       // Shuttle 2
       "DB_OPC_Machine".Parameters.Presence.Shuttle2UndrilledPart := "DB_PartManagement".sPosition.sShuttle2.Undrilled.Presence.Part;
       "DB_OPC_Machine".Parameters.Presence.Shuttle2UndrilledBw := "DB_PartManagement".sPosition.sShuttle2.Undrilled.Presence.BW;
       "DB_OPC_Machine".Parameters.Presence.Shuttle2DrilledPart := "DB_PartManagement".sPosition.sShuttle2.Drilled.Presence.Part;
       "DB_OPC_Machine".Parameters.Presence.Shuttle2DrilledBw := "DB_PartManagement".sPosition.sShuttle2.Drilled.Presence.BW;

       // Gripper
       "DB_OPC_Machine".Parameters.Presence.GripperUndrilledPart := "DB_PartManagement".sPosition.sGripper.Undrilled.Presence.Part;
       "DB_OPC_Machine".Parameters.Presence.GripperUndrilledBw := "DB_PartManagement".sPosition.sGripper.Undrilled.Presence.BW;
       "DB_OPC_Machine".Parameters.Presence.GripperDrilledPart := "DB_PartManagement".sPosition.sGripper.Drilled.Presence.Part;
       "DB_OPC_Machine".Parameters.Presence.GripperDrilledBw := "DB_PartManagement".sPosition.sGripper.Drilled.Presence.BW;

       // Fixture
       "DB_OPC_Machine".Parameters.Presence.FixtureUndrilledPart := "DB_PartManagement".sPosition.sFixture.Undrilled.Presence.Part;
       "DB_OPC_Machine".Parameters.Presence.FixtureUndrilledBw := "DB_PartManagement".sPosition.sFixture.Undrilled.Presence.BW;
       "DB_OPC_Machine".Parameters.Presence.FixtureDrilledPart := "DB_PartManagement".sPosition.sFixture.Drilled.Presence.Part;
       "DB_OPC_Machine".Parameters.Presence.FixtureDrilledBw := "DB_PartManagement".sPosition.sFixture.Drilled.Presence.BW;
   END_REGION

   REGION Presence V2
       // // Shuttle 1
       // #sPresenceShuttle1UndrilledPart("HMI_Change Enable" := #sHmiChangeEnable,
       //                                 ioPLC_State := "DB_PartManagement".sPosition.sShuttle1.Undrilled.Presence.Part,
       //                                 ioHMI_State := "DB_OPC_Machine".Parameters.Presence.Shuttle1UndrilledPart);

       // #sPresenceShuttle1UndrilledBw("HMI_Change Enable" := #sHmiChangeEnable,
       //                               ioPLC_State := "DB_PartManagement".sPosition.sShuttle1.Undrilled.Presence.BW,
       //                               ioHMI_State := "DB_OPC_Machine".Parameters.Presence.Shuttle1UndrilledBw);

       // #sPresenceShuttle1DrilledPart("HMI_Change Enable" := #sHmiChangeEnable,
       //                                 ioPLC_State := "DB_PartManagement".sPosition.sShuttle1.Drilled.Presence.Part,
       //                                 ioHMI_State := "DB_OPC_Machine".Parameters.Presence.Shuttle1DrilledPart);

       // #sPresenceShuttle1DrilledBw("HMI_Change Enable" := #sHmiChangeEnable,
       //                               ioPLC_State := "DB_PartManagement".sPosition.sShuttle1.Drilled.Presence.BW,
       //                               ioHMI_State := "DB_OPC_Machine".Parameters.Presence.Shuttle1DrilledBw);

       //  // Shuttle 2
       //  #sPresenceShuttle2UndrilledPart("HMI_Change Enable" := #sHmiChangeEnable,
       //                                  ioPLC_State := "DB_PartManagement".sPosition.sShuttle2.Undrilled.Presence.Part,
       //                                  ioHMI_State := "DB_OPC_Machine".Parameters.Presence.Shuttle2UndrilledPart);

       //  #sPresenceShuttle2UndrilledBw("HMI_Change Enable" := #sHmiChangeEnable,
       //                                ioPLC_State := "DB_PartManagement".sPosition.sShuttle2.Undrilled.Presence.BW,
       //                                ioHMI_State := "DB_OPC_Machine".Parameters.Presence.Shuttle2UndrilledBw);

       //  #sPresenceShuttle2DrilledPart("HMI_Change Enable" := #sHmiChangeEnable,
       //                                ioPLC_State := "DB_PartManagement".sPosition.sShuttle2.Drilled.Presence.Part,
       //                                ioHMI_State := "DB_OPC_Machine".Parameters.Presence.Shuttle2DrilledPart);

       //  #sPresenceShuttle2DrilledBw("HMI_Change Enable" := #sHmiChangeEnable,
       //                              ioPLC_State := "DB_PartManagement".sPosition.sShuttle2.Drilled.Presence.BW,
       //                              ioHMI_State := "DB_OPC_Machine".Parameters.Presence.Shuttle2DrilledBw);

       //  // Gripper
       //  #sPresenceGripperUndrilledPart("HMI_Change Enable" := #sHmiChangeEnable,
       //                                 ioPLC_State := "DB_PartManagement".sPosition.sGripper.Undrilled.Presence.Part,
       //                                 ioHMI_State := "DB_OPC_Machine".Parameters.Presence.GripperUndrilledPart);

       //  #sPresenceGripperUndrilledBw("HMI_Change Enable" := #sHmiChangeEnable,
       //                               ioPLC_State := "DB_PartManagement".sPosition.sGripper.Undrilled.Presence.BW,
       //                               ioHMI_State := "DB_OPC_Machine".Parameters.Presence.GripperUndrilledBw);

       //  #sPresenceGripperDrilledPart("HMI_Change Enable" := #sHmiChangeEnable,
       //                               ioPLC_State := "DB_PartManagement".sPosition.sGripper.Drilled.Presence.Part,
       //                               ioHMI_State := "DB_OPC_Machine".Parameters.Presence.GripperDrilledPart);

       //  #sPresenceGripperDrilledBw("HMI_Change Enable" := #sHmiChangeEnable,
       //                             ioPLC_State := "DB_PartManagement".sPosition.sGripper.Drilled.Presence.BW,
       //                             ioHMI_State := "DB_OPC_Machine".Parameters.Presence.GripperDrilledBw);

       //  // Fixture
       //  #sPresenceFixtureUndrilledPart("HMI_Change Enable" := #sHmiChangeEnable,
       //                                 ioPLC_State := "DB_PartManagement".sPosition.sFixture.Undrilled.Presence.Part,
       //                                 ioHMI_State := "DB_OPC_Machine".Parameters.Presence.FixtureUndrilledPart);

       //  #sPresenceFixtureUndrilledBw("HMI_Change Enable" := #sHmiChangeEnable,
       //                               ioPLC_State := "DB_PartManagement".sPosition.sFixture.Undrilled.Presence.BW,
       //                               ioHMI_State := "DB_OPC_Machine".Parameters.Presence.FixtureUndrilledBw);

       //  #sPresenceFixtureDrilledPart("HMI_Change Enable" := #sHmiChangeEnable,
       //                               ioPLC_State := "DB_PartManagement".sPosition.sFixture.Drilled.Presence.Part,
       //                               ioHMI_State := "DB_OPC_Machine".Parameters.Presence.FixtureDrilledPart);

       //  #sPresenceFixtureDrilledBw("HMI_Change Enable" := #sHmiChangeEnable,
       //                             ioPLC_State := "DB_PartManagement".sPosition.sFixture.Drilled.Presence.BW,
       //                             ioHMI_State := "DB_OPC_Machine".Parameters.Presence.FixtureDrilledBw);
   END_REGION
END_FUNCTION_BLOCK

FUNCTION_BLOCK "FB_HMI_PLC_Pos"   // FB80, SCL
{ S7_Optimized_Access := 'TRUE' }
// stored: MemoryReserve 100, SetENOAutomatically false
   VAR_INPUT
      "HMI_Change Enable" : Bool;
   END_VAR
   VAR_IN_OUT
      ioPLC_State : Bool;
      ioHMI_State : Bool;
   END_VAR
   VAR
      PLC_StateMemo : Bool;
      HMI_StateMemo : Bool;
   END_VAR
BEGIN
   REGION Description header 
       //==================================================================================
       // POSALUX Swiss SA / (C) Copyright 2026
       //----------------------------------------------------------------------------------
       // Title: FB_HMI_PLC_Pos
       // Comment/Function: 
       // Author: Fabien WALDT
       // Engineering: TIA Portal v20
       //----------------------------------------------------------------------------------
       // Change log table:
       // Version  | Date     | Expert in charge | Changes applied
       // ---------|----------|------------------|-----------------------------------------
       // 00.00.01 | 20260521 | WFA              | First released version
       // =================================================================================
   END_REGION

   REGION Update Values
       IF #ioPLC_State <> #PLC_StateMemo OR NOT #"HMI_Change Enable" THEN
           #ioHMI_State := #ioPLC_State;
           #HMI_StateMemo := #ioPLC_State;
           #PLC_StateMemo := #ioPLC_State;
       ELSIF (#ioHMI_State <> #HMI_StateMemo) AND #"HMI_Change Enable" THEN
           #ioPLC_State := #ioHMI_State;
           #PLC_StateMemo := #ioHMI_State;
           #HMI_StateMemo := #ioHMI_State;
       END_IF;

   END_REGION
END_FUNCTION_BLOCK

FUNCTION_BLOCK "FB_OPC_AxisManagement"   // FB60, SCL
{ S7_Optimized_Access := 'TRUE' }
// stored: MemoryReserve 100, SetENOAutomatically false
   VAR
      sTeachButton : "FB_HmiKeysSignals";
      sAxisToTeachIndex { S7_SetPoint := 'True'} : DInt;
      sPositionToTeachIndex : DInt;
      sError { ExternalAccessible := 'False'; ExternalVisible := 'False'; ExternalWritable := 'False'} : Bool;
      sDone { ExternalAccessible := 'False'; ExternalVisible := 'False'; ExternalWritable := 'False'} : Bool;
      sState { ExternalAccessible := 'False'; ExternalVisible := 'False'; ExternalWritable := 'False'} : Word;
      sReadGUD_X_Load : "LBP_ReadGUD";
      sReadGUD_X_Unload { S7_SetPoint := 'True'} : "LBP_ReadGUD";
      sReadGUD_X_Blowing { S7_SetPoint := 'True'} : "LBP_ReadGUD";
      sReadGUD_Y_Load : "LBP_ReadGUD";
      sReadGUD_Y_Unload { S7_SetPoint := 'True'} : "LBP_ReadGUD";
      sReadGUD_Y_Blowing { S7_SetPoint := 'True'} : "LBP_ReadGUD";
      sReadGUD_B_Load : "LBP_ReadGUD";
      sReadGUD_B_Unload { S7_SetPoint := 'True'} : "LBP_ReadGUD";
      sReadGUD_B_Blowing { S7_SetPoint := 'True'} : "LBP_ReadGUD";
      sReadGUD_ZM_Safe { S7_SetPoint := 'True'} : "LBP_ReadGUD";
      sReadGUD_ZL_Safe { S7_SetPoint := 'True'} : "LBP_ReadGUD";
      sVarName { S7_SetPoint := 'True'} : String;
      sTON_On : TON_TIME;
      sTON_OFF { S7_SetPoint := 'True'} : TON_TIME;
      sPulseReadGUD { S7_SetPoint := 'True'} : Bool;
      sID : Int;
   END_VAR
   VAR_TEMP
      tIndex : Int;
   END_VAR
   VAR CONSTANT
      U1_AXIS_ID : DInt := 111;
      U2_AXIS_ID : DInt := 112;
      V_AXIS_ID : DInt := 120;
      W_AXIS_ID : DInt := 130;
      X_AXIS_ID : DInt := 210;
      Y_AXIS_ID : DInt := 220;
      ZL_AXIS_ID : DInt := 230;
      ZM_AXIS_ID : DInt := 240;
      B_AXIS_ID : DInt := 320;
      EXTERNAL_LOADER_ID : DInt := 211;
      SEMI_AUTO_ID : DInt := 212;
      EXT_OF_SAFETY_GATE_EXT_ID : DInt := 221;
      INT_OF_SAFETY_GATE_EXT_ID : DInt := 222;
      INSIDE_SAFETY_GATE_ID : DInt := 223;
      EXT_OF_SAFETY_GATE_INT_ID : DInt := 224;
      INT_OF_SAFETY_GATE_INT_ID : DInt := 225;
      PART_DETECTOR_ID : DInt := 230;
      BACKWALL_LOAD_ID : DInt := 241;
      BACKWALL_UNLOAD_ID : DInt := 242;
      BACKWALL_DETECTOR_ID : DInt := 250;
      LOADER_BLOW_TO_SHUTTLE_ID : DInt := 260;
      LOADER_BLOW_TO_SHUTTLE_1_ID : DInt := 261;
      LOADER_BLOW_TO_SHUTTLE_2_ID : DInt := 262;
      FROM_SHUTTLE_TO_LOADER_ID : DInt := 310;
      FROM_SHUTTLE_1_TO_LOADER : DInt := 311;
      FROM_SHUTTLE_2_TO_LOADER : DInt := 312;
      SAFE : DInt := 400;
      APPROACH_SHUTTLE_1 : DInt := 421;
      APPROACH_SHUTTLE_2 : DInt := 422;
      APPROACH_WORK_CLAMP : DInt := 430;
      FROM_LOADER_TO_WORK : DInt := 610;
      FROM_WORK_TO_LOADER : DInt := 620;
      LOADER_BLOW_TO_WORK : DInt := 730;
      STATION1 : Byte := 1;
   END_VAR
BEGIN
   REGION Description header 
       //==================================================================================
       // POSALUX Swiss SA / (C) Copyright 2025
       //----------------------------------------------------------------------------------
       // Title: FB_OPC_AxisManagement
       // Comment/Function: 
       // Author: Fabien WALDT
       // Engineering: TIA Portal v20
       //----------------------------------------------------------------------------------
       // Change log table:
       // Version  | Date     | Expert in charge | Changes applied
       // ---------|----------|------------------|-----------------------------------------
       // 00.00.01 | 20260109 | WFA              | First released version
       // =================================================================================
   END_REGION
   REGION Axis - Actual Values
       // Number of axis
       "DB_OPC_Axis".ActualValues.NumberOfAxes := 9;

       // Axis01_X
       #sID := 1;
       "DB_OPC_Axis".ActualValues.Axes[#sID].ActualPosition := "DB_AxisPosition".sAxis01_X."$AA_IM";
       "DB_OPC_Axis".ActualValues.Axes[#sID].AxisId := #X_AXIS_ID;
       "DB_OPC_Axis".ActualValues.Axes[#sID].StationNumber := #STATION1;
       // Axis02_Y
       #sID := #sID + 1;
       "DB_OPC_Axis".ActualValues.Axes[#sID].ActualPosition := "DB_AxisPosition".sAxis02_Y."$AA_IM";
       "DB_OPC_Axis".ActualValues.Axes[#sID].AxisId := #Y_AXIS_ID;
       "DB_OPC_Axis".ActualValues.Axes[#sID].StationNumber := #STATION1;
       // Axis03_ZM
       #sID := #sID + 1;
       "DB_OPC_Axis".ActualValues.Axes[#sID].ActualPosition := "DB_AxisPosition".sAxis03_ZM."$AA_IM";
       "DB_OPC_Axis".ActualValues.Axes[#sID].AxisId := #ZM_AXIS_ID;
       "DB_OPC_Axis".ActualValues.Axes[#sID].StationNumber := #STATION1;
       // Axis04_B
       #sID := #sID + 1;
       "DB_OPC_Axis".ActualValues.Axes[#sID].ActualPosition := "DB_AxisPosition".sAxis04_B."$AA_IM";
       "DB_OPC_Axis".ActualValues.Axes[#sID].AxisId := #B_AXIS_ID;
       "DB_OPC_Axis".ActualValues.Axes[#sID].StationNumber := #STATION1;
       // Axis05_U1
       #sID := #sID + 1;
       "DB_OPC_Axis".ActualValues.Axes[#sID].ActualPosition := "DB_AxisPosition".sAxis05_U1."$AA_IM";
       "DB_OPC_Axis".ActualValues.Axes[#sID].AxisId := #U1_AXIS_ID;
       "DB_OPC_Axis".ActualValues.Axes[#sID].StationNumber := #STATION1;
       // Axis06_U2
       #sID := #sID + 1;
       "DB_OPC_Axis".ActualValues.Axes[#sID].ActualPosition := "DB_AxisPosition".sAxis06_U2."$AA_IM";
       "DB_OPC_Axis".ActualValues.Axes[#sID].AxisId := #U2_AXIS_ID;
       "DB_OPC_Axis".ActualValues.Axes[#sID].StationNumber := #STATION1;
       // Axis07_V
       #sID := #sID + 1;
       "DB_OPC_Axis".ActualValues.Axes[#sID].ActualPosition := "DB_AxisPosition".sAxis07_V."$AA_IM";
       "DB_OPC_Axis".ActualValues.Axes[#sID].AxisId := #V_AXIS_ID;
       "DB_OPC_Axis".ActualValues.Axes[#sID].StationNumber := #STATION1;
       // Axis08_W
       #sID := #sID + 1;
       "DB_OPC_Axis".ActualValues.Axes[#sID].ActualPosition := "DB_AxisPosition".sAxis08_W."$AA_IM";
       "DB_OPC_Axis".ActualValues.Axes[#sID].AxisId := #W_AXIS_ID;
       "DB_OPC_Axis".ActualValues.Axes[#sID].StationNumber := #STATION1;
       // Axis09_ZL
       #sID := #sID + 1;
       "DB_OPC_Axis".ActualValues.Axes[#sID].ActualPosition := "DB_AxisPosition".sAxis09_ZL."$AA_IM";
       "DB_OPC_Axis".ActualValues.Axes[#sID].AxisId := #ZL_AXIS_ID;
       "DB_OPC_Axis".ActualValues.Axes[#sID].StationNumber := #STATION1;
   END_REGION

   REGION Taught Position PLC
       // Number of items
       "DB_OPC_Axis".TaughtPositions.NumberOfItems := 48;

       REGION Axis05_U1
           // External loader
           #sID := 1;
           "DB_OPC_Axis".TaughtPositions.Items[#sID].AxisId := #U1_AXIS_ID;
           "DB_OPC_Axis".TaughtPositions.Items[#sID].PositionId := #EXTERNAL_LOADER_ID;
           "DB_OPC_Axis".TaughtPositions.Items[#sID].StationNumber := #STATION1;
           "DB_OPC_Axis".TaughtPositions.Items[#sID].Value := "DB_AxisPosMachinePLC".Axis_U1.ExtLoadUnloadAuto;
           // Semi-auto
           #sID := #sID + 1;
           "DB_OPC_Axis".TaughtPositions.Items[#sID].AxisId := #U1_AXIS_ID;
           "DB_OPC_Axis".TaughtPositions.Items[#sID].PositionId := #SEMI_AUTO_ID;
           "DB_OPC_Axis".TaughtPositions.Items[#sID].StationNumber := #STATION1;
           "DB_OPC_Axis".TaughtPositions.Items[#sID].Value := "DB_AxisPosMachinePLC".Axis_U1.ExtLoadUnloadManu;
           // Ext of safety gate ext
           #sID := #sID + 1;
           "DB_OPC_Axis".TaughtPositions.Items[#sID].AxisId := #U1_AXIS_ID;
           "DB_OPC_Axis".TaughtPositions.Items[#sID].PositionId := #EXT_OF_SAFETY_GATE_EXT_ID;
           "DB_OPC_Axis".TaughtPositions.Items[#sID].StationNumber := #STATION1;
           "DB_OPC_Axis".TaughtPositions.Items[#sID].Value := "DB_AxisPosMachinePLC".Axis_U1.ExtGateExt;
           // Int of safety gate ext
           #sID := #sID + 1;
           "DB_OPC_Axis".TaughtPositions.Items[#sID].AxisId := #U1_AXIS_ID;
           "DB_OPC_Axis".TaughtPositions.Items[#sID].PositionId := #INT_OF_SAFETY_GATE_EXT_ID;
           "DB_OPC_Axis".TaughtPositions.Items[#sID].StationNumber := #STATION1;
           "DB_OPC_Axis".TaughtPositions.Items[#sID].Value := "DB_AxisPosMachinePLC".Axis_U1.IntGateExt;
           // Inside safety gate
           #sID := #sID + 1;
           "DB_OPC_Axis".TaughtPositions.Items[#sID].AxisId := #U1_AXIS_ID;
           "DB_OPC_Axis".TaughtPositions.Items[#sID].PositionId := #INSIDE_SAFETY_GATE_ID;
           "DB_OPC_Axis".TaughtPositions.Items[#sID].StationNumber := #STATION1;
           "DB_OPC_Axis".TaughtPositions.Items[#sID].Value := "DB_AxisPosMachinePLC".Axis_U1.Sas;
           // Ext of safety gate Int
           #sID := #sID + 1;
           "DB_OPC_Axis".TaughtPositions.Items[#sID].AxisId := #U1_AXIS_ID;
           "DB_OPC_Axis".TaughtPositions.Items[#sID].PositionId := #EXT_OF_SAFETY_GATE_INT_ID;
           "DB_OPC_Axis".TaughtPositions.Items[#sID].StationNumber := #STATION1;
           "DB_OPC_Axis".TaughtPositions.Items[#sID].Value := "DB_AxisPosMachinePLC".Axis_U1.ExtGateInt;
           // Int of safety gate Int
           #sID := #sID + 1;
           "DB_OPC_Axis".TaughtPositions.Items[#sID].AxisId := #U1_AXIS_ID;
           "DB_OPC_Axis".TaughtPositions.Items[#sID].PositionId := #INT_OF_SAFETY_GATE_INT_ID;
           "DB_OPC_Axis".TaughtPositions.Items[#sID].StationNumber := #STATION1;
           "DB_OPC_Axis".TaughtPositions.Items[#sID].Value := "DB_AxisPosMachinePLC".Axis_U1.IntGateInt;
           // Part detector
           #sID := #sID + 1;
           "DB_OPC_Axis".TaughtPositions.Items[#sID].AxisId := #U1_AXIS_ID;
           "DB_OPC_Axis".TaughtPositions.Items[#sID].PositionId := #PART_DETECTOR_ID;
           "DB_OPC_Axis".TaughtPositions.Items[#sID].StationNumber := #STATION1;
           "DB_OPC_Axis".TaughtPositions.Items[#sID].Value := "DB_AxisPosMachinePLC".Axis_U1.PartControl;
           // Backwall load
           #sID := #sID + 1;
           "DB_OPC_Axis".TaughtPositions.Items[#sID].AxisId := #U1_AXIS_ID;
           "DB_OPC_Axis".TaughtPositions.Items[#sID].PositionId := #BACKWALL_LOAD_ID;
           "DB_OPC_Axis".TaughtPositions.Items[#sID].StationNumber := #STATION1;
           "DB_OPC_Axis".TaughtPositions.Items[#sID].Value := "DB_AxisPosMachinePLC".Axis_U1.BwLoad;
           // Backwall unload
           #sID := #sID + 1;
           "DB_OPC_Axis".TaughtPositions.Items[#sID].AxisId := #U1_AXIS_ID;
           "DB_OPC_Axis".TaughtPositions.Items[#sID].PositionId := #BACKWALL_UNLOAD_ID;
           "DB_OPC_Axis".TaughtPositions.Items[#sID].StationNumber := #STATION1;
           "DB_OPC_Axis".TaughtPositions.Items[#sID].Value := "DB_AxisPosMachinePLC".Axis_U1.BwUnLoad;
           // Backwall detector
           #sID := #sID + 1;
           "DB_OPC_Axis".TaughtPositions.Items[#sID].AxisId := #U1_AXIS_ID;
           "DB_OPC_Axis".TaughtPositions.Items[#sID].PositionId := #BACKWALL_DETECTOR_ID;
           "DB_OPC_Axis".TaughtPositions.Items[#sID].StationNumber := #STATION1;
           "DB_OPC_Axis".TaughtPositions.Items[#sID].Value := "DB_AxisPosMachinePLC".Axis_U1.BwControl;
           // Loader blow to shuttle
           #sID := #sID + 1;
           "DB_OPC_Axis".TaughtPositions.Items[#sID].AxisId := #U1_AXIS_ID;
           "DB_OPC_Axis".TaughtPositions.Items[#sID].PositionId := #LOADER_BLOW_TO_SHUTTLE_ID;
           "DB_OPC_Axis".TaughtPositions.Items[#sID].StationNumber := #STATION1;
           "DB_OPC_Axis".TaughtPositions.Items[#sID].Value := "DB_AxisPosMachinePLC".Axis_U1.Blowing;
           // From shuttle to Loader
           #sID := #sID + 1;
           "DB_OPC_Axis".TaughtPositions.Items[#sID].AxisId := #U1_AXIS_ID;
           "DB_OPC_Axis".TaughtPositions.Items[#sID].PositionId := #FROM_SHUTTLE_TO_LOADER_ID;
           "DB_OPC_Axis".TaughtPositions.Items[#sID].StationNumber := #STATION1;
           "DB_OPC_Axis".TaughtPositions.Items[#sID].Value := "DB_AxisPosMachinePLC".Axis_U1.IntLoadUnload;
       END_REGION

       REGION Axis06_U2
           // External loader
           #sID := #sID + 1;
           "DB_OPC_Axis".TaughtPositions.Items[#sID].AxisId := #U2_AXIS_ID;
           "DB_OPC_Axis".TaughtPositions.Items[#sID].PositionId := #EXTERNAL_LOADER_ID;
           "DB_OPC_Axis".TaughtPositions.Items[#sID].StationNumber := #STATION1;
           "DB_OPC_Axis".TaughtPositions.Items[#sID].Value := "DB_AxisPosMachinePLC".Axis_U2.ExtLoadUnloadAuto;
           // Semi-auto
           #sID := #sID + 1;
           "DB_OPC_Axis".TaughtPositions.Items[#sID].AxisId := #U2_AXIS_ID;
           "DB_OPC_Axis".TaughtPositions.Items[#sID].PositionId := #SEMI_AUTO_ID;
           "DB_OPC_Axis".TaughtPositions.Items[#sID].StationNumber := #STATION1;
           "DB_OPC_Axis".TaughtPositions.Items[#sID].Value := "DB_AxisPosMachinePLC".Axis_U2.ExtLoadUnloadManu;
           // Ext of safety gate ext
           #sID := #sID + 1;
           "DB_OPC_Axis".TaughtPositions.Items[#sID].AxisId := #U2_AXIS_ID;
           "DB_OPC_Axis".TaughtPositions.Items[#sID].PositionId := #EXT_OF_SAFETY_GATE_EXT_ID;
           "DB_OPC_Axis".TaughtPositions.Items[#sID].StationNumber := #STATION1;
           "DB_OPC_Axis".TaughtPositions.Items[#sID].Value := "DB_AxisPosMachinePLC".Axis_U2.ExtGateExt;
           // Int of safety gate ext
           #sID := #sID + 1;
           "DB_OPC_Axis".TaughtPositions.Items[#sID].AxisId := #U2_AXIS_ID;
           "DB_OPC_Axis".TaughtPositions.Items[#sID].PositionId := #INT_OF_SAFETY_GATE_EXT_ID;
           "DB_OPC_Axis".TaughtPositions.Items[#sID].StationNumber := #STATION1;
           "DB_OPC_Axis".TaughtPositions.Items[#sID].Value := "DB_AxisPosMachinePLC".Axis_U2.IntGateExt;
           // Inside safety gate
           #sID := #sID + 1;
           "DB_OPC_Axis".TaughtPositions.Items[#sID].AxisId := #U2_AXIS_ID;
           "DB_OPC_Axis".TaughtPositions.Items[#sID].PositionId := #INSIDE_SAFETY_GATE_ID;
           "DB_OPC_Axis".TaughtPositions.Items[#sID].StationNumber := #STATION1;
           "DB_OPC_Axis".TaughtPositions.Items[#sID].Value := "DB_AxisPosMachinePLC".Axis_U2.Sas;
           // Ext of safety gate Int
           #sID := #sID + 1;
           "DB_OPC_Axis".TaughtPositions.Items[#sID].AxisId := #U2_AXIS_ID;
           "DB_OPC_Axis".TaughtPositions.Items[#sID].PositionId := #EXT_OF_SAFETY_GATE_INT_ID;
           "DB_OPC_Axis".TaughtPositions.Items[#sID].StationNumber := #STATION1;
           "DB_OPC_Axis".TaughtPositions.Items[#sID].Value := "DB_AxisPosMachinePLC".Axis_U2.ExtGateInt;
           // Int of safety gate Int
           #sID := #sID + 1;
           "DB_OPC_Axis".TaughtPositions.Items[#sID].AxisId := #U2_AXIS_ID;
           "DB_OPC_Axis".TaughtPositions.Items[#sID].PositionId := #INT_OF_SAFETY_GATE_INT_ID;
           "DB_OPC_Axis".TaughtPositions.Items[#sID].StationNumber := #STATION1;
           "DB_OPC_Axis".TaughtPositions.Items[#sID].Value := "DB_AxisPosMachinePLC".Axis_U2.IntGateInt;
           // Part detector
           #sID := #sID + 1;
           "DB_OPC_Axis".TaughtPositions.Items[#sID].AxisId := #U2_AXIS_ID;
           "DB_OPC_Axis".TaughtPositions.Items[#sID].PositionId := #PART_DETECTOR_ID;
           "DB_OPC_Axis".TaughtPositions.Items[#sID].StationNumber := #STATION1;
           "DB_OPC_Axis".TaughtPositions.Items[#sID].Value := "DB_AxisPosMachinePLC".Axis_U2.PartControl;
           // Backwall load
           #sID := #sID + 1;
           "DB_OPC_Axis".TaughtPositions.Items[#sID].AxisId := #U2_AXIS_ID;
           "DB_OPC_Axis".TaughtPositions.Items[#sID].PositionId := #BACKWALL_LOAD_ID;
           "DB_OPC_Axis".TaughtPositions.Items[#sID].StationNumber := #STATION1;
           "DB_OPC_Axis".TaughtPositions.Items[#sID].Value := "DB_AxisPosMachinePLC".Axis_U2.BwLoad;
           // Backwall unload
           #sID := #sID + 1;
           "DB_OPC_Axis".TaughtPositions.Items[#sID].AxisId := #U2_AXIS_ID;
           "DB_OPC_Axis".TaughtPositions.Items[#sID].PositionId := #BACKWALL_UNLOAD_ID;
           "DB_OPC_Axis".TaughtPositions.Items[#sID].StationNumber := #STATION1;
           "DB_OPC_Axis".TaughtPositions.Items[#sID].Value := "DB_AxisPosMachinePLC".Axis_U2.BwUnLoad;
           // Backwall detector
           #sID := #sID + 1;
           "DB_OPC_Axis".TaughtPositions.Items[#sID].AxisId := #U2_AXIS_ID;
           "DB_OPC_Axis".TaughtPositions.Items[#sID].PositionId := #BACKWALL_DETECTOR_ID;
           "DB_OPC_Axis".TaughtPositions.Items[#sID].StationNumber := #STATION1;
           "DB_OPC_Axis".TaughtPositions.Items[#sID].Value := "DB_AxisPosMachinePLC".Axis_U2.BwControl;
           // Loader blow to shuttle
           #sID := #sID + 1;
           "DB_OPC_Axis".TaughtPositions.Items[#sID].AxisId := #U2_AXIS_ID;
           "DB_OPC_Axis".TaughtPositions.Items[#sID].PositionId := #LOADER_BLOW_TO_SHUTTLE_ID;
           "DB_OPC_Axis".TaughtPositions.Items[#sID].StationNumber := #STATION1;
           "DB_OPC_Axis".TaughtPositions.Items[#sID].Value := "DB_AxisPosMachinePLC".Axis_U2.Blowing;
           // From shuttle to Loader
           #sID := #sID + 1;
           "DB_OPC_Axis".TaughtPositions.Items[#sID].AxisId := #U2_AXIS_ID;
           "DB_OPC_Axis".TaughtPositions.Items[#sID].PositionId := #FROM_SHUTTLE_TO_LOADER_ID;
           "DB_OPC_Axis".TaughtPositions.Items[#sID].StationNumber := #STATION1;
           "DB_OPC_Axis".TaughtPositions.Items[#sID].Value := "DB_AxisPosMachinePLC".Axis_U2.IntLoadUnload;
       END_REGION

       REGION Axis07_V
           // Loader blow to shuttle 1
           #sID := #sID + 1;
           "DB_OPC_Axis".TaughtPositions.Items[#sID].AxisId := #V_AXIS_ID;
           "DB_OPC_Axis".TaughtPositions.Items[#sID].PositionId := #LOADER_BLOW_TO_SHUTTLE_1_ID;
           "DB_OPC_Axis".TaughtPositions.Items[#sID].StationNumber := #STATION1;
           "DB_OPC_Axis".TaughtPositions.Items[#sID].Value := "DB_AxisPosMachinePLC".Axis_V.Shuttle_1.Blowing;
           // Loader blow to shuttle 2
           #sID := #sID + 1;
           "DB_OPC_Axis".TaughtPositions.Items[#sID].AxisId := #V_AXIS_ID;
           "DB_OPC_Axis".TaughtPositions.Items[#sID].PositionId := #LOADER_BLOW_TO_SHUTTLE_2_ID;
           "DB_OPC_Axis".TaughtPositions.Items[#sID].StationNumber := #STATION1;
           "DB_OPC_Axis".TaughtPositions.Items[#sID].Value := "DB_AxisPosMachinePLC".Axis_V.Shuttle_2.Blowing;
           // From shuttle 1 to loader
           #sID := #sID + 1;
           "DB_OPC_Axis".TaughtPositions.Items[#sID].AxisId := #V_AXIS_ID;
           "DB_OPC_Axis".TaughtPositions.Items[#sID].PositionId := #FROM_SHUTTLE_1_TO_LOADER;
           "DB_OPC_Axis".TaughtPositions.Items[#sID].StationNumber := #STATION1;
           "DB_OPC_Axis".TaughtPositions.Items[#sID].Value := "DB_AxisPosMachinePLC".Axis_V.Shuttle_1.LoadUnload;
           // From shuttle 2 to loader
           #sID := #sID + 1;
           "DB_OPC_Axis".TaughtPositions.Items[#sID].AxisId := #V_AXIS_ID;
           "DB_OPC_Axis".TaughtPositions.Items[#sID].PositionId := #FROM_SHUTTLE_2_TO_LOADER;
           "DB_OPC_Axis".TaughtPositions.Items[#sID].StationNumber := #STATION1;
           "DB_OPC_Axis".TaughtPositions.Items[#sID].Value := "DB_AxisPosMachinePLC".Axis_V.Shuttle_2.LoadUnload;
           // Safe
           #sID := #sID + 1;
           "DB_OPC_Axis".TaughtPositions.Items[#sID].AxisId := #V_AXIS_ID;
           "DB_OPC_Axis".TaughtPositions.Items[#sID].PositionId := #SAFE;
           "DB_OPC_Axis".TaughtPositions.Items[#sID].StationNumber := #STATION1;
           "DB_OPC_Axis".TaughtPositions.Items[#sID].Value := "DB_AxisPosMachinePLC".Axis_V.Safe;
       END_REGION

       REGION Axis08_W
           // Loader blow to shuttle 1
           #sID := #sID + 1;
           "DB_OPC_Axis".TaughtPositions.Items[#sID].AxisId := #W_AXIS_ID;
           "DB_OPC_Axis".TaughtPositions.Items[#sID].PositionId := #LOADER_BLOW_TO_SHUTTLE_1_ID;
           "DB_OPC_Axis".TaughtPositions.Items[#sID].StationNumber := #STATION1;
           "DB_OPC_Axis".TaughtPositions.Items[#sID].Value := "DB_AxisPosMachinePLC".Axis_W.Shuttle_1.Blowing;
           // Loader blow to shuttle 2
           #sID := #sID + 1;
           "DB_OPC_Axis".TaughtPositions.Items[#sID].AxisId := #W_AXIS_ID;
           "DB_OPC_Axis".TaughtPositions.Items[#sID].PositionId := #LOADER_BLOW_TO_SHUTTLE_2_ID;
           "DB_OPC_Axis".TaughtPositions.Items[#sID].StationNumber := #STATION1;
           "DB_OPC_Axis".TaughtPositions.Items[#sID].Value := "DB_AxisPosMachinePLC".Axis_W.Shuttle_2.Blowing;
           // From shuttle 1 to loader
           #sID := #sID + 1;
           "DB_OPC_Axis".TaughtPositions.Items[#sID].AxisId := #W_AXIS_ID;
           "DB_OPC_Axis".TaughtPositions.Items[#sID].PositionId := #FROM_SHUTTLE_1_TO_LOADER;
           "DB_OPC_Axis".TaughtPositions.Items[#sID].StationNumber := #STATION1;
           "DB_OPC_Axis".TaughtPositions.Items[#sID].Value := "DB_AxisPosMachinePLC".Axis_W.Shuttle_1.LoadUnload;
           // From shuttle 2 to loader
           #sID := #sID + 1;
           "DB_OPC_Axis".TaughtPositions.Items[#sID].AxisId := #W_AXIS_ID;
           "DB_OPC_Axis".TaughtPositions.Items[#sID].PositionId := #FROM_SHUTTLE_2_TO_LOADER;
           "DB_OPC_Axis".TaughtPositions.Items[#sID].StationNumber := #STATION1;
           "DB_OPC_Axis".TaughtPositions.Items[#sID].Value := "DB_AxisPosMachinePLC".Axis_W.Shuttle_2.LoadUnload;
           // Safe
           #sID := #sID + 1;
           "DB_OPC_Axis".TaughtPositions.Items[#sID].AxisId := #W_AXIS_ID;
           "DB_OPC_Axis".TaughtPositions.Items[#sID].PositionId := #SAFE;
           "DB_OPC_Axis".TaughtPositions.Items[#sID].StationNumber := #STATION1;
           "DB_OPC_Axis".TaughtPositions.Items[#sID].Value := "DB_AxisPosMachinePLC".Axis_W.Safe;
       END_REGION

       REGION Axis07_V (Fixture)
           // From loader to work
           #sID := #sID + 1;
           "DB_OPC_Axis".TaughtPositions.Items[#sID].AxisId := #V_AXIS_ID;
           "DB_OPC_Axis".TaughtPositions.Items[#sID].PositionId := #FROM_LOADER_TO_WORK;
           "DB_OPC_Axis".TaughtPositions.Items[#sID].StationNumber := #STATION1;
           "DB_OPC_Axis".TaughtPositions.Items[#sID].Value := "DB_AxisPosMachinePLC".Axis_V.Fixture.Load;
           // From work to loader
           #sID := #sID + 1;
           "DB_OPC_Axis".TaughtPositions.Items[#sID].AxisId := #V_AXIS_ID;
           "DB_OPC_Axis".TaughtPositions.Items[#sID].PositionId := #FROM_WORK_TO_LOADER;
           "DB_OPC_Axis".TaughtPositions.Items[#sID].StationNumber := #STATION1;
           "DB_OPC_Axis".TaughtPositions.Items[#sID].Value := "DB_AxisPosMachinePLC".Axis_V.Fixture.Unload;
           // Loader blow to work
           #sID := #sID + 1;
           "DB_OPC_Axis".TaughtPositions.Items[#sID].AxisId := #V_AXIS_ID;
           "DB_OPC_Axis".TaughtPositions.Items[#sID].PositionId := #LOADER_BLOW_TO_WORK;
           "DB_OPC_Axis".TaughtPositions.Items[#sID].StationNumber := #STATION1;
           "DB_OPC_Axis".TaughtPositions.Items[#sID].Value := "DB_AxisPosMachinePLC".Axis_V.Fixture.Blowing;
       END_REGION

       REGION Axis08_W (Fixture)
           // Approach work clamp NOT USED
           // #sID := #sID + 1;
           // "DB_OPC_Axis".TaughtPositions.Items[#sID].AxisId := #W_AXIS_ID;
           // "DB_OPC_Axis".TaughtPositions.Items[#sID].PositionId := #APPROACH_WORK_CLAMP;
           // "DB_OPC_Axis".TaughtPositions.Items[#sID].StationNumber := #STATION1;
           // "DB_OPC_Axis".TaughtPositions.Items[#sID].Value := "DB_AxisPosMachineNC".Axis_W.Approach;
           // From loader to work
           #sID := #sID + 1;
           "DB_OPC_Axis".TaughtPositions.Items[#sID].AxisId := #W_AXIS_ID;
           "DB_OPC_Axis".TaughtPositions.Items[#sID].PositionId := #FROM_LOADER_TO_WORK;
           "DB_OPC_Axis".TaughtPositions.Items[#sID].StationNumber := #STATION1;
           "DB_OPC_Axis".TaughtPositions.Items[#sID].Value := "DB_AxisPosMachinePLC".Axis_W.Fixture.Load;
           // From work to loader
           #sID := #sID + 1;
           "DB_OPC_Axis".TaughtPositions.Items[#sID].AxisId := #W_AXIS_ID;
           "DB_OPC_Axis".TaughtPositions.Items[#sID].PositionId := #FROM_WORK_TO_LOADER;
           "DB_OPC_Axis".TaughtPositions.Items[#sID].StationNumber := #STATION1;
           "DB_OPC_Axis".TaughtPositions.Items[#sID].Value := "DB_AxisPosMachinePLC".Axis_W.Fixture.Unload;
           // Loader blow to work
           #sID := #sID + 1;
           "DB_OPC_Axis".TaughtPositions.Items[#sID].AxisId := #W_AXIS_ID;
           "DB_OPC_Axis".TaughtPositions.Items[#sID].PositionId := #LOADER_BLOW_TO_WORK;
           "DB_OPC_Axis".TaughtPositions.Items[#sID].StationNumber := #STATION1;
           "DB_OPC_Axis".TaughtPositions.Items[#sID].Value := "DB_AxisPosMachinePLC".Axis_W.Fixture.Blowing;
       END_REGION
   END_REGION

   REGION Taught Position NC
       REGION Axis01_X
           // From loader to work
           #sID := #sID + 1;
           "DB_OPC_Axis".TaughtPositions.Items[#sID].AxisId := #X_AXIS_ID;
           "DB_OPC_Axis".TaughtPositions.Items[#sID].PositionId := #FROM_LOADER_TO_WORK;
           "DB_OPC_Axis".TaughtPositions.Items[#sID].StationNumber := #STATION1;
           "DB_OPC_Axis".TaughtPositions.Items[#sID].Value := "DB_AxisPosMachineNC".Axis_X.Load;
           // From work to loader
           #sID := #sID + 1;
           "DB_OPC_Axis".TaughtPositions.Items[#sID].AxisId := #X_AXIS_ID;
           "DB_OPC_Axis".TaughtPositions.Items[#sID].PositionId := #FROM_WORK_TO_LOADER;
           "DB_OPC_Axis".TaughtPositions.Items[#sID].StationNumber := #STATION1;
           "DB_OPC_Axis".TaughtPositions.Items[#sID].Value := "DB_AxisPosMachineNC".Axis_X.Unload;
           // Loader blow to work
           #sID := #sID + 1;
           "DB_OPC_Axis".TaughtPositions.Items[#sID].AxisId := #X_AXIS_ID;
           "DB_OPC_Axis".TaughtPositions.Items[#sID].PositionId := #LOADER_BLOW_TO_WORK;
           "DB_OPC_Axis".TaughtPositions.Items[#sID].StationNumber := #STATION1;
           "DB_OPC_Axis".TaughtPositions.Items[#sID].Value := "DB_AxisPosMachineNC".Axis_X.Blowing;
       END_REGION

       REGION Axis02_Y
           // From loader to work
           #sID := #sID + 1;
           "DB_OPC_Axis".TaughtPositions.Items[#sID].AxisId := #Y_AXIS_ID;
           "DB_OPC_Axis".TaughtPositions.Items[#sID].PositionId := #FROM_LOADER_TO_WORK;
           "DB_OPC_Axis".TaughtPositions.Items[#sID].StationNumber := #STATION1;
           "DB_OPC_Axis".TaughtPositions.Items[#sID].Value := "DB_AxisPosMachineNC".Axis_Y.Load;
           // From work to loader
           #sID := #sID + 1;
           "DB_OPC_Axis".TaughtPositions.Items[#sID].AxisId := #Y_AXIS_ID;
           "DB_OPC_Axis".TaughtPositions.Items[#sID].PositionId := #FROM_WORK_TO_LOADER;
           "DB_OPC_Axis".TaughtPositions.Items[#sID].StationNumber := #STATION1;
           "DB_OPC_Axis".TaughtPositions.Items[#sID].Value := "DB_AxisPosMachineNC".Axis_Y.Unload;
           // Loader blow to work
           #sID := #sID + 1;
           "DB_OPC_Axis".TaughtPositions.Items[#sID].AxisId := #Y_AXIS_ID;
           "DB_OPC_Axis".TaughtPositions.Items[#sID].PositionId := #LOADER_BLOW_TO_WORK;
           "DB_OPC_Axis".TaughtPositions.Items[#sID].StationNumber := #STATION1;
           "DB_OPC_Axis".TaughtPositions.Items[#sID].Value := "DB_AxisPosMachineNC".Axis_Y.Blowing;
       END_REGION

       // REGION Axis04_B Not Used
       //     // From loader to work
       //     #sID := #sID + 1;
       //     "DB_OPC_Axis".TaughtPositions.Items[#sID].AxisId := #B_AXIS_ID;
       //     "DB_OPC_Axis".TaughtPositions.Items[#sID].PositionId := #FROM_LOADER_TO_WORK;
       //     "DB_OPC_Axis".TaughtPositions.Items[#sID].StationNumber := #STATION1;
       //     "DB_OPC_Axis".TaughtPositions.Items[#sID].Value := "DB_AxisPosMachineNC".Axis_B.Load;
       //     // From work to loader
       //     #sID := #sID + 1;
       //     "DB_OPC_Axis".TaughtPositions.Items[#sID].AxisId := #B_AXIS_ID;
       //     "DB_OPC_Axis".TaughtPositions.Items[#sID].PositionId := #FROM_WORK_TO_LOADER;
       //     "DB_OPC_Axis".TaughtPositions.Items[#sID].StationNumber := #STATION1;
       //     "DB_OPC_Axis".TaughtPositions.Items[#sID].Value := "DB_AxisPosMachineNC".Axis_B.Unload;
       //     // Loader blow to work
       //     #sID := #sID + 1;
       //     "DB_OPC_Axis".TaughtPositions.Items[#sID].AxisId := #B_AXIS_ID;
       //     "DB_OPC_Axis".TaughtPositions.Items[#sID].PositionId := #LOADER_BLOW_TO_WORK;
       //     "DB_OPC_Axis".TaughtPositions.Items[#sID].StationNumber := #STATION1;
       //     "DB_OPC_Axis".TaughtPositions.Items[#sID].Value := "DB_AxisPosMachineNC".Axis_B.Blowing;
       // END_REGION


   END_REGION

   REGION Teach
       // Call button
       #sTeachButton(ioOPC := "DB_OPC_Axis".Teach.Buttons.Teach);
       #sTeachButton.sKeyDisable := "LBP_ModeGroup".E_JOG;
       #sTeachButton.sLedSWStatus := #sTeachButton.sKeySWToggleStatus;

       // Search axis index
       #sAxisToTeachIndex := 0;
       "DB_OPC_Axis".Teach.Current.ActualPosition := 0.0;
       FOR #tIndex := 1 TO "DB_OPC_Axis".ActualValues.NumberOfAxes DO
           IF "DB_OPC_Axis".ActualValues.Axes[#tIndex].AxisId = "DB_OPC_Axis".Teach.Parameters.AxisId THEN
               #sAxisToTeachIndex := #tIndex;
               "DB_OPC_Axis".Teach.Current.ActualPosition := "DB_OPC_Axis".ActualValues.Axes[#sAxisToTeachIndex].ActualPosition;
           END_IF;
       END_FOR;
       // Search position index
       #sPositionToTeachIndex := 0;
       "DB_OPC_Axis".Teach.Current.TaughtPosition := 0.0;
       FOR #tIndex := 1 TO "DB_OPC_Axis".TaughtPositions.NumberOfItems DO
           IF "DB_OPC_Axis".TaughtPositions.Items[#tIndex].AxisId = "DB_OPC_Axis".Teach.Parameters.AxisId
               AND "DB_OPC_Axis".TaughtPositions.Items[#tIndex].PositionId = "DB_OPC_Axis".Teach.Parameters.PositionId THEN
               #sPositionToTeachIndex := #tIndex;
               "DB_OPC_Axis".Teach.Current.TaughtPosition := "DB_OPC_Axis".TaughtPositions.Items[#sPositionToTeachIndex].Value;
           END_IF;
       END_FOR;

       // // If Teach Button, Copy Axis ActualPosition to TaughtPosition 
       // IF #TeachButton.KeySWToggleStatus THEN
       //     "DB_OPC_Axis".TaughtPositions.Items[#PositionToTeachIndex].Value := "DB_OPC_Axis".ActualValues.Axes[#AxisToTeachIndex].ActualPosition;
       //     #TeachButton.KeySWToggleStatus := FALSE;
       // END_IF;
   END_REGION

   REGION Copy Current values to Taught Values
       IF #sTeachButton.sKeySWToggleStatus THEN
           CASE "DB_OPC_Axis".Teach.Parameters.AxisId OF
           #U1_AXIS_ID:
               CASE "DB_OPC_Axis".Teach.Parameters.PositionId OF
                   #EXTERNAL_LOADER_ID:
                       "DB_AxisPosMachinePLC".Axis_U1.ExtLoadUnloadAuto := "DB_AxisPosition".sAxis05_U1."$AA_IM";
                   #SEMI_AUTO_ID:
                       "DB_AxisPosMachinePLC".Axis_U1.ExtLoadUnloadManu := "DB_AxisPosition".sAxis05_U1."$AA_IM";
                   #EXT_OF_SAFETY_GATE_EXT_ID:
                       "DB_AxisPosMachinePLC".Axis_U1.ExtGateExt := "DB_AxisPosition".sAxis05_U1."$AA_IM";
                   #INT_OF_SAFETY_GATE_EXT_ID:
                       "DB_AxisPosMachinePLC".Axis_U1.IntGateExt := "DB_AxisPosition".sAxis05_U1."$AA_IM";
                   #INSIDE_SAFETY_GATE_ID:
                       "DB_AxisPosMachinePLC".Axis_U1.Sas := "DB_AxisPosition".sAxis05_U1."$AA_IM";
                   #EXT_OF_SAFETY_GATE_INT_ID:
                       "DB_AxisPosMachinePLC".Axis_U1.ExtGateInt := "DB_AxisPosition".sAxis05_U1."$AA_IM";
                   #INT_OF_SAFETY_GATE_INT_ID:
                       "DB_AxisPosMachinePLC".Axis_U1.IntGateInt := "DB_AxisPosition".sAxis05_U1."$AA_IM";
                   #PART_DETECTOR_ID:
                       "DB_AxisPosMachinePLC".Axis_U1.PartControl := "DB_AxisPosition".sAxis05_U1."$AA_IM";
                   #BACKWALL_LOAD_ID:
                       "DB_AxisPosMachinePLC".Axis_U1.BwLoad := "DB_AxisPosition".sAxis05_U1."$AA_IM";
                   #BACKWALL_UNLOAD_ID:
                       "DB_AxisPosMachinePLC".Axis_U1.BwUnLoad := "DB_AxisPosition".sAxis05_U1."$AA_IM";
                   #BACKWALL_DETECTOR_ID:
                       "DB_AxisPosMachinePLC".Axis_U1.BwControl := "DB_AxisPosition".sAxis05_U1."$AA_IM";
                   #LOADER_BLOW_TO_SHUTTLE_ID:
                       "DB_AxisPosMachinePLC".Axis_U1.Blowing := "DB_AxisPosition".sAxis05_U1."$AA_IM";
                   #FROM_SHUTTLE_TO_LOADER_ID:
                       "DB_AxisPosMachinePLC".Axis_U1.IntLoadUnload := "DB_AxisPosition".sAxis05_U1."$AA_IM";
               END_CASE;
           #U2_AXIS_ID:
               CASE "DB_OPC_Axis".Teach.Parameters.PositionId OF
                   #EXTERNAL_LOADER_ID:
                       "DB_AxisPosMachinePLC".Axis_U1.ExtLoadUnloadAuto := "DB_AxisPosition".sAxis06_U2."$AA_IM";
                   #SEMI_AUTO_ID:
                       "DB_AxisPosMachinePLC".Axis_U1.ExtLoadUnloadManu := "DB_AxisPosition".sAxis06_U2."$AA_IM";
                   #EXT_OF_SAFETY_GATE_EXT_ID:
                       "DB_AxisPosMachinePLC".Axis_U1.ExtGateExt := "DB_AxisPosition".sAxis06_U2."$AA_IM";
                   #INT_OF_SAFETY_GATE_EXT_ID:
                       "DB_AxisPosMachinePLC".Axis_U1.IntGateExt := "DB_AxisPosition".sAxis06_U2."$AA_IM";
                   #INSIDE_SAFETY_GATE_ID:
                       "DB_AxisPosMachinePLC".Axis_U1.Sas := "DB_AxisPosition".sAxis06_U2."$AA_IM";
                   #EXT_OF_SAFETY_GATE_INT_ID:
                       "DB_AxisPosMachinePLC".Axis_U1.ExtGateInt := "DB_AxisPosition".sAxis06_U2."$AA_IM";
                   #INT_OF_SAFETY_GATE_INT_ID:
                       "DB_AxisPosMachinePLC".Axis_U1.IntGateInt := "DB_AxisPosition".sAxis06_U2."$AA_IM";
                   #PART_DETECTOR_ID:
                       "DB_AxisPosMachinePLC".Axis_U1.PartControl := "DB_AxisPosition".sAxis06_U2."$AA_IM";
                   #BACKWALL_LOAD_ID:
                       "DB_AxisPosMachinePLC".Axis_U1.BwLoad := "DB_AxisPosition".sAxis06_U2."$AA_IM";
                   #BACKWALL_UNLOAD_ID:
                       "DB_AxisPosMachinePLC".Axis_U1.BwUnLoad := "DB_AxisPosition".sAxis06_U2."$AA_IM";
                   #BACKWALL_DETECTOR_ID:
                       "DB_AxisPosMachinePLC".Axis_U1.BwControl := "DB_AxisPosition".sAxis06_U2."$AA_IM";
                   #LOADER_BLOW_TO_SHUTTLE_ID:
                       "DB_AxisPosMachinePLC".Axis_U1.Blowing := "DB_AxisPosition".sAxis06_U2."$AA_IM";
                   #FROM_SHUTTLE_TO_LOADER_ID:
                       "DB_AxisPosMachinePLC".Axis_U1.IntLoadUnload := "DB_AxisPosition".sAxis06_U2."$AA_IM";
               END_CASE;
           #V_AXIS_ID:
               CASE "DB_OPC_Axis".Teach.Parameters.PositionId OF
                   #LOADER_BLOW_TO_SHUTTLE_1_ID:
                       "DB_AxisPosMachinePLC".Axis_V.Shuttle_1.Blowing := "DB_AxisPosition".sAxis07_V."$AA_IM";
                   #LOADER_BLOW_TO_SHUTTLE_2_ID:
                       "DB_AxisPosMachinePLC".Axis_V.Shuttle_2.Blowing := "DB_AxisPosition".sAxis07_V."$AA_IM";
                   #FROM_SHUTTLE_1_TO_LOADER:
                       "DB_AxisPosMachinePLC".Axis_V.Shuttle_1.LoadUnload := "DB_AxisPosition".sAxis07_V."$AA_IM";
                   #FROM_SHUTTLE_2_TO_LOADER:
                       "DB_AxisPosMachinePLC".Axis_V.Shuttle_2.LoadUnload := "DB_AxisPosition".sAxis07_V."$AA_IM";
                   #SAFE:
                       "DB_AxisPosMachinePLC".Axis_V.Safe := "DB_AxisPosition".sAxis07_V."$AA_IM";

                   #FROM_LOADER_TO_WORK:
                       "DB_AxisPosMachinePLC".Axis_V.Fixture.Load := "DB_AxisPosition".sAxis07_V."$AA_IM";
                   #FROM_WORK_TO_LOADER:
                       "DB_AxisPosMachinePLC".Axis_V.Fixture.Unload := "DB_AxisPosition".sAxis07_V."$AA_IM";
                   #LOADER_BLOW_TO_WORK:
                       "DB_AxisPosMachinePLC".Axis_V.Fixture.Blowing := "DB_AxisPosition".sAxis07_V."$AA_IM";
               END_CASE;
           #W_AXIS_ID:
               CASE "DB_OPC_Axis".Teach.Parameters.PositionId OF
                   #LOADER_BLOW_TO_SHUTTLE_1_ID:
                       "DB_AxisPosMachinePLC".Axis_W.Shuttle_1.Blowing := "DB_AxisPosition".sAxis08_W."$AA_IM";
                   #LOADER_BLOW_TO_SHUTTLE_2_ID:
                       "DB_AxisPosMachinePLC".Axis_W.Shuttle_2.Blowing := "DB_AxisPosition".sAxis08_W."$AA_IM";
                   #FROM_SHUTTLE_1_TO_LOADER:
                       "DB_AxisPosMachinePLC".Axis_W.Shuttle_1.LoadUnload := "DB_AxisPosition".sAxis08_W."$AA_IM";
                   #FROM_SHUTTLE_2_TO_LOADER:
                       "DB_AxisPosMachinePLC".Axis_W.Shuttle_2.LoadUnload := "DB_AxisPosition".sAxis08_W."$AA_IM";
                   #SAFE:
                       "DB_AxisPosMachinePLC".Axis_W.Safe := "DB_AxisPosition".sAxis08_W."$AA_IM";

                   #FROM_LOADER_TO_WORK:
                       "DB_AxisPosMachinePLC".Axis_V.Fixture.Load := "DB_AxisPosition".sAxis08_W."$AA_IM";
                   #FROM_WORK_TO_LOADER:
                       "DB_AxisPosMachinePLC".Axis_V.Fixture.Unload := "DB_AxisPosition".sAxis08_W."$AA_IM";
                   #LOADER_BLOW_TO_WORK:
                       "DB_AxisPosMachinePLC".Axis_V.Fixture.Blowing := "DB_AxisPosition".sAxis08_W."$AA_IM";
               END_CASE;
           #X_AXIS_ID:
               CASE "DB_OPC_Axis".Teach.Parameters.PositionId OF
                   #FROM_LOADER_TO_WORK:
                       "DB_AxisPosMachineNC".Axis_X.Load := "DB_AxisPosition".sAxis01_X."$AA_IM";
                   #FROM_WORK_TO_LOADER:
                       "DB_AxisPosMachineNC".Axis_X.Unload := "DB_AxisPosition".sAxis01_X."$AA_IM";
                   #LOADER_BLOW_TO_WORK:
                       "DB_AxisPosMachineNC".Axis_X.Blowing := "DB_AxisPosition".sAxis01_X."$AA_IM";
               END_CASE;
           #Y_AXIS_ID:
               CASE "DB_OPC_Axis".Teach.Parameters.PositionId OF
                   #FROM_LOADER_TO_WORK:
                       "DB_AxisPosMachineNC".Axis_X.Load := "DB_AxisPosition".sAxis02_Y."$AA_IM";
                   #FROM_WORK_TO_LOADER:
                       "DB_AxisPosMachineNC".Axis_X.Unload := "DB_AxisPosition".sAxis02_Y."$AA_IM";
                   #LOADER_BLOW_TO_WORK:
                       "DB_AxisPosMachineNC".Axis_X.Blowing := "DB_AxisPosition".sAxis02_Y."$AA_IM";
               END_CASE;
           #B_AXIS_ID:
               CASE "DB_OPC_Axis".Teach.Parameters.PositionId OF
                   #FROM_LOADER_TO_WORK:
                       "DB_AxisPosMachineNC".Axis_X.Load := "DB_AxisPosition".sAxis04_B."$AA_IM";
                   #FROM_WORK_TO_LOADER:
                       "DB_AxisPosMachineNC".Axis_X.Unload := "DB_AxisPosition".sAxis04_B."$AA_IM";
                   #LOADER_BLOW_TO_WORK:
                       "DB_AxisPosMachineNC".Axis_X.Blowing := "DB_AxisPosition".sAxis04_B."$AA_IM";
               END_CASE;
       END_CASE;
       #sTeachButton.sKeySWToggleStatus := FALSE;
     END_IF;
   END_REGION

   REGION Read NC Position

       // TON phase ON (5 secondes)
       #sTON_On(
              IN := #sPulseReadGUD,
              PT := T#5s);

       // TON phase OFF (5 secondes)
       #sTON_OFF(
               IN := NOT #sPulseReadGUD,
               PT := T#5s);

      IF #sTON_On.Q THEN
           #sPulseReadGUD := FALSE;
       END_IF;

       IF #sTON_OFF.Q THEN
           #sPulseReadGUD := TRUE;
       END_IF;


       REGION X Axis
           #sVarName := 'CH_X_LOAD';

           #sReadGUD_X_Load(Req := #sPulseReadGUD,
                           Addr := #sVarName,
                           Area := 2,
                           Unit := 1,
                           Index1 := 0,
                           Index2 := 0,
                           CnvtToken := FALSE,
                           VarToken := NULL,
                           Error => #sReadGUD_X_Load.Error,
                           Done => #sReadGUD_X_Load.Done,
                           State => #sReadGUD_X_Load.State,
                           RD := "DB_AxisPosMachineNC".Axis_X.Load);

           #sVarName := 'CH_X_UNLOAD';

           #sReadGUD_X_Unload(Req := #sPulseReadGUD,
                           Addr := #sVarName,
                           Area := 2,
                           Unit := 1,
                           Index1 := 0,
                           Index2 := 0,
                           CnvtToken := FALSE,
                           VarToken := NULL,
                           Error => #sReadGUD_X_Unload.Error,
                           Done => #sReadGUD_X_Unload.Done,
                           State => #sReadGUD_X_Unload.State,
                           RD := "DB_AxisPosMachineNC".Axis_X.Unload);

           #sVarName := 'CH_X_BLOW';

           #sReadGUD_X_Blowing(Req := #sPulseReadGUD,
                                  Addr := #sVarName,
                                  Area := 2,
                                  Unit := 1,
                                  Index1 := 0,
                                  Index2 := 0,
                                  CnvtToken := FALSE,
                                  VarToken := NULL,
                                  Error => #sReadGUD_X_Blowing.Error,
                                  Done => #sReadGUD_X_Blowing.Done,
                                  State => #sReadGUD_X_Blowing.State,
                                  RD := "DB_AxisPosMachineNC".Axis_X.Blowing);
       END_REGION
       REGION Y Axis
           #sVarName := 'CH_Y_LOAD';

           #sReadGUD_Y_Load(Req := NOT #sPulseReadGUD,
                           Addr := #sVarName,
                           Area := 2,
                           Unit := 1,
                           Index1 := 0,
                           Index2 := 0,
                           CnvtToken := FALSE,
                           VarToken := NULL,
                           Error => #sReadGUD_Y_Load.Error,
                           Done => #sReadGUD_Y_Load.Done,
                           State => #sReadGUD_Y_Load.State,
                           RD := "DB_AxisPosMachineNC".Axis_Y.Load);

           #sVarName := 'CH_Y_UNLOAD';

           #sReadGUD_Y_Unload(Req := NOT #sPulseReadGUD,
                             Addr := #sVarName,
                             Area := 2,
                             Unit := 1,
                             Index1 := 0,
                             Index2 := 0,
                             CnvtToken := FALSE,
                             VarToken := NULL,
                             Error => #sReadGUD_Y_Unload.Error,
                             Done => #sReadGUD_Y_Unload.Done,
                             State => #sReadGUD_Y_Unload.State,
                             RD := "DB_AxisPosMachineNC".Axis_Y.Unload);

           #sVarName := 'CH_Y_BLOW';

           #sReadGUD_Y_Blowing(Req := NOT #sPulseReadGUD,
                              Addr := #sVarName,
                              Area := 2,
                              Unit := 1,
                              Index1 := 0,
                              Index2 := 0,
                              CnvtToken := FALSE,
                              VarToken := NULL,
                              Error => #sReadGUD_Y_Blowing.Error,
                              Done => #sReadGUD_Y_Blowing.Done,
                              State => #sReadGUD_Y_Blowing.State,
                              RD := "DB_AxisPosMachineNC".Axis_Y.Blowing);
       END_REGION
       REGION B Axis
           #sVarName := 'CH_B_LOAD';

           #sReadGUD_B_Load(Req := #sPulseReadGUD,
                           Addr := #sVarName,
                           Area := 2,
                           Unit := 1,
                           Index1 := 0,
                           Index2 := 0,
                           CnvtToken := FALSE,
                           VarToken := NULL,
                           Error => #sReadGUD_B_Load.Error,
                           Done => #sReadGUD_B_Load.Done,
                           State => #sReadGUD_B_Load.State,
                           RD := "DB_AxisPosMachineNC".Axis_B.Load);

           #sVarName := 'CH_B_UNLOAD';

           #sReadGUD_B_Unload(Req := #sPulseReadGUD,
                             Addr := #sVarName,
                             Area := 2,
                             Unit := 1,
                             Index1 := 0,
                             Index2 := 0,
                             CnvtToken := FALSE,
                             VarToken := NULL,
                             Error => #sReadGUD_B_Unload.Error,
                             Done => #sReadGUD_B_Unload.Done,
                             State => #sReadGUD_B_Unload.State,
                             RD := "DB_AxisPosMachineNC".Axis_B.Unload);

           #sVarName := 'CH_B_BLOW';

           #sReadGUD_B_Blowing(Req := #sPulseReadGUD,
                              Addr := #sVarName,
                              Area := 2,
                              Unit := 1,
                              Index1 := 0,
                              Index2 := 0,
                              CnvtToken := FALSE,
                              VarToken := NULL,
                              Error => #sReadGUD_B_Blowing.Error,
                              Done => #sReadGUD_B_Blowing.Done,
                              State => #sReadGUD_B_Blowing.State,
                              RD := "DB_AxisPosMachineNC".Axis_B.Blowing);
       END_REGION
       REGION ZM Axis
           #sVarName := 'CH_ZM_SAFE';

           #sReadGUD_ZM_Safe(Req := #sPulseReadGUD,
                              Addr := #sVarName,
                              Area := 2,
                              Unit := 1,
                              Index1 := 0,
                              Index2 := 0,
                              CnvtToken := FALSE,
                              VarToken := NULL,
                              Error => #sReadGUD_ZM_Safe.Error,
                              Done => #sReadGUD_ZM_Safe.Done,
                              State => #sReadGUD_ZM_Safe.State,
                              RD := "DB_AxisPosMachineNC".Axis_ZM.Safe);
         END_REGION

         REGION ZL Axis
             #sVarName := 'CH_ZL_SAFE';

             #sReadGUD_ZL_Safe(Req := NOT #sPulseReadGUD,
                              Addr := #sVarName,
                              Area := 2,
                              Unit := 1,
                              Index1 := 0,
                              Index2 := 0,
                              CnvtToken := FALSE,
                              VarToken := NULL,
                              Error => #sReadGUD_ZL_Safe.Error,
                              Done => #sReadGUD_ZL_Safe.Done,
                              State => #sReadGUD_ZL_Safe.State,
                              RD := "DB_AxisPosMachineNC".Axis_ZL.Safe);
         END_REGION
   END_REGION
END_FUNCTION_BLOCK

FUNCTION_BLOCK "FB_HmiKeysSignals"   // FB812, SCL
{ S7_Optimized_Access := 'TRUE' }
// stored: AutoNumber false, MemoryReserve 100, SetENOAutomatically false
   VAR_IN_OUT
      ioOPC : "UDT_OPC_Button";
   END_VAR
   VAR
      sKeySWStatus : Bool;
      sKeySWToggleStatus : Bool;
      sKeyDisable : Bool;
      sKeySWPositiveFront : Bool;
      sKeySWNegativeFront : Bool;
      sKeySWTogglePositiveFront : Bool;
      sKeySWToggleNegativeFront : Bool;
      sLedSWStatus : Bool;
      sLedSWStatusBlink : Bool;
      sRT_KeySWPositiveFront { S7_SetPoint := 'True'} : R_TRIG;
      sFT_KeySWNegativeFront { S7_SetPoint := 'True'} : F_TRIG;
      sRT_KeySWTogglePositiveFront { S7_SetPoint := 'True'} : R_TRIG;
      sFT_KeySWToggleNegativeFront { S7_SetPoint := 'True'} : F_TRIG;
   END_VAR
BEGIN
   REGION Description header 
       //==================================================================================
       // POSALUX Swiss SA / (C) Copyright 2025
       //----------------------------------------------------------------------------------
       // Title: FB_HmiKeysSignals 
       // Comment/Function: 
       //
       // Author: Fabien Waldt
       // Engineering: TIA Portal v19
       //----------------------------------------------------------------------------------
       // Change log table:
       // Version  | Date     | Expert in charge | Changes applied
       // ---------|----------|------------------|------------------------------------
       // 00.00.01 | 20250911 | WFA              | First released version
       // ==================================================================================
   END_REGION

   REGION Key Enable
       #ioOPC.bEnable := NOT #sKeyDisable;
   END_REGION

   REGION Inputs keys
       // Management of the software input
       IF NOT #sKeyDisable THEN
           #sKeySWStatus := #ioOPC.bClick;
       // ELSE
       //     #sKeySWStatus := FALSE;
       //     #sKeySWToggleStatus := FALSE;
       END_IF;

       // Reset KeyOPCStatus (bClick from HMI)
       #ioOPC.bClick := FALSE;

       // Rising/falling edge detection when pressing the button
       #sRT_KeySWPositiveFront(CLK := #sKeySWStatus,
                              Q => #sKeySWPositiveFront);

       #sFT_KeySWNegativeFront(CLK := #sKeySWStatus,
                              Q => #sKeySWNegativeFront);

       // Toggle state update
       IF #sKeySWPositiveFront THEN
           #sKeySWToggleStatus := NOT #sKeySWToggleStatus;
       END_IF;

       // Rising/falling edge detection of the toggle state
       #sRT_KeySWTogglePositiveFront(CLK := #sKeySWToggleStatus,
                                    Q => #sKeySWTogglePositiveFront);

       #sFT_KeySWToggleNegativeFront(CLK := #sKeySWToggleStatus,
                                    Q => #sKeySWToggleNegativeFront);
   END_REGION

   REGION Outputs LED   
       #ioOPC.bIsPressed := #sLedSWStatus;

       // Blink Status
       #ioOPC.bBlink := #sLedSWStatusBlink;
   END_REGION
END_FUNCTION_BLOCK

FUNCTION_BLOCK "FB_OPC_State"   // FB75, SCL
{ S7_Optimized_Access := 'TRUE' }
// stored: MemoryReserve 100, SetENOAutomatically false
   VAR
      sAutoReq : Bool;
      sSemiAutoReq : Bool;
      sManuReq : Bool;
      sRT_AutoReq : R_TRIG;
      sRT_SemiAutoReq : R_TRIG;
      sRT_ManuReq : R_TRIG;
   END_VAR
   VAR CONSTANT
      AUTO : Byte := 1;
      SEMI_AUTO : Byte := 2;
      MANU : Byte := 3;
      UNDEFINED : Byte := 0;
   END_VAR
BEGIN
   REGION Description header 
       //==================================================================================
       // POSALUX Swiss SA / (C) Copyright 2024
       //----------------------------------------------------------------------------------
       // Title: 
       // Comment/Function: 
       //
       // Author: Fabien WALDT
       // Engineering: TIA Portal v20
       //----------------------------------------------------------------------------------
       // Change log table:
       // Version  | Date     | Expert in charge | Changes applied
       // ---------|----------|------------------|------------------------------------
       // 00.00.01 | 20260130 | WFA              | First released version
       // ==================================================================================
   END_REGION

   REGION Current
       // CanLockDoor
       "DB_OPC_Machine".State.Current.CanLockDoor := "LBP_ModeGroup".E_JOG
       AND "DB_DigitalInputs".sFrontDoorClosed.sSWStatus;

       // CanUnlockDoor
       "DB_OPC_Machine".State.Current.CanUnlockDoor := "LBP_ModeGroup".E_JOG
       AND "DB_DigitalInputs".sFrontDoorLocked.sSWStatus;

       // LoadingMode
       // 1 = Auto
       // 2 = Semi Auto
       // 3 = Manu 
       IF "DB_WorkingModes".sAuto THEN
           "DB_OPC_Machine".State.Current.LoadingMode := #AUTO;
       ELSIF "DB_WorkingModes".sSemiAuto THEN
           "DB_OPC_Machine".State.Current.LoadingMode := #SEMI_AUTO;
       ELSIF "DB_WorkingModes".sManu THEN
           "DB_OPC_Machine".State.Current.LoadingMode := #MANU;
       ELSE
           "DB_OPC_Machine".State.Current.LoadingMode := #UNDEFINED;
       END_IF;

       // IsDoorLocked
       "DB_OPC_Machine".State.Current.IsDoorLocked := "DB_DigitalInputs".sFrontDoorLocked.sSWStatus;

       // IsEmptying
       "DB_OPC_Machine".State.Current.IsEmptying := "DB_WorkingModes".sEmptying;

       // IsInitialized
       "DB_OPC_Machine".State.Current.IsInitialized := "DB_PowerOn".sMachineReadySoft;

       // IsRunning
       "DB_OPC_Machine".State.Current.IsRunning := "LBP_Chan1".E_ProgRunning;
   END_REGION

   REGION
       // Request Change Mode
       IF "DB_OPC_Machine".State.Requests.LoadingMode.RequestChangeMode THEN
           IF "DB_OPC_Machine".State.Requests.LoadingMode.TargetMode = #AUTO THEN
               #sAutoReq := TRUE;
           ELSIF "DB_OPC_Machine".State.Requests.LoadingMode.TargetMode = #SEMI_AUTO THEN
               #sSemiAutoReq := TRUE;
           ELSIF "DB_OPC_Machine".State.Requests.LoadingMode.TargetMode = #MANU THEN
               #sManuReq := TRUE;
           END_IF;
           "DB_OPC_Machine".State.Requests.LoadingMode.RequestChangeMode := FALSE;
           "DB_OPC_Machine".State.Requests.LoadingMode.TargetMode := #UNDEFINED;
       END_IF;

       #sRT_AutoReq(CLK := #sAutoReq);
       #sRT_SemiAutoReq(CLK := #sSemiAutoReq);
       #sRT_ManuReq(CLK := #sManuReq);

       // Request Lock Door
       IF "DB_OPC_Machine".State.Requests.RequestLockDoor THEN
           "DB_HMISetting".LockDoorReq := TRUE;
           "DB_OPC_Machine".State.Requests.RequestLockDoor := FALSE;
       END_IF;

       // Request Start Auto
       IF "DB_OPC_Machine".State.Requests.RequestStartAuto THEN
           "DB_HMISetting".StartAutoReq := TRUE;
           "DB_OPC_Machine".State.Requests.RequestStartAuto := FALSE;
       END_IF;

       // Request Start Emptying
       IF "DB_OPC_Machine".State.Requests.RequestStartEmptying THEN
           "DB_HMISetting".WorkingMode.EmptyingReq := TRUE;
           "DB_OPC_Machine".State.Requests.RequestStartEmptying := FALSE;
       END_IF;

       // Request Stop Auto
       IF "DB_OPC_Machine".State.Requests.RequestStopAuto THEN
           "DB_HMISetting".StopAutoReq := TRUE;
           "DB_OPC_Machine".State.Requests.RequestStopAuto := FALSE;
       END_IF;

       // Request Stop Emptying (Back to Normal Mode)
       IF "DB_OPC_Machine".State.Requests.RequestStopEmptying THEN
           "DB_HMISetting".WorkingMode.EmptyingReq := FALSE;
       END_IF;
       "DB_OPC_Machine".State.Requests.RequestStopEmptying := FALSE;

       // Request Unlock Door
       IF "DB_OPC_Machine".State.Requests.RequestUnlockDoor THEN
           "DB_HMISetting".UnlockDoorReq := TRUE;
           "DB_OPC_Machine".State.Requests.RequestUnlockDoor := FALSE;
       END_IF;
   END_REGION

   REGION CNCMode
       IF "LBP_ModeGroup".E_AUTO THEN
           "DB_OPC_Machine".State.Current.CncMode := 1;
       ELSIF "LBP_ModeGroup".E_JOG THEN
           "DB_OPC_Machine".State.Current.CncMode := 2;
       ELSIF "LBP_ModeGroup".E_MDA THEN
           "DB_OPC_Machine".State.Current.CncMode := 3;
       ELSE
           "DB_OPC_Machine".State.Current.CncMode := 0;
       END_IF;
   END_REGION

   REGION MachineOverride
       "DB_OPC_Machine".State.Current.MachineOverride := "DB_FeedOverride".oFeedOverride;
   END_REGION
END_FUNCTION_BLOCK

FUNCTION_BLOCK "FB_RealTime"   // FB74, SCL
{ S7_Optimized_Access := 'TRUE' }
// stored: MemoryReserve 100, SetENOAutomatically false
BEGIN
   REGION Description header 
       //==================================================================================
       // POSALUX Swiss SA / (C) Copyright 2024
       //----------------------------------------------------------------------------------
       // Title: FB_RealTime
       // Comment/Function: 
       //
       // Author: Fabien WALDT
       // Engineering: TIA Portal v20
       //----------------------------------------------------------------------------------
       // Change log table:
       // Version  | Date     | Expert in charge | Changes applied
       // ---------|----------|------------------|------------------------------------
       // 00.00.01 | 20260127 | WFA              | First released version
       // ==================================================================================
   END_REGION

   REGION Digital Inputs
       "DB_OPC_RealTime".X_AxisBrakePressCtrl := "DB_DigitalInputs".sX_AxisBrakePressCtrl.sSWStatus;
       "DB_OPC_RealTime".Y_AxisBrakePressCtrl := "DB_DigitalInputs".sY_AxisBrakePressCtrl.sSWStatus;
       "DB_OPC_RealTime".BreakerCtrl := "DB_DigitalInputs".sBreakerCtrl.sSWStatus;
       "DB_OPC_RealTime".CabinetTemperatureCtrl := "DB_DigitalInputs".sCabinetTemperatureCtrl.sSWStatus;
       "DB_OPC_RealTime".UpsPowerFailure := "DB_DigitalInputs".sUPS_PowerFailure.sSWStatus;
       "DB_OPC_RealTime".AirPressureCtrl := "DB_DigitalInputs".sAirPressureCtrl.sSWStatus;
       "DB_OPC_RealTime".ShutterClosed := "DB_DigitalInputs".sShutterClosed.sSWStatus;
       "DB_OPC_RealTime".AirDryerOK := "DB_DigitalInputs".sAirDryerOK.sSWStatus;
       "DB_OPC_RealTime".UPS_BatteryOK := "DB_DigitalInputs".sUPS_BatteryOK.sSWStatus;
       "DB_OPC_RealTime".FrontDoorClosed := "DB_DigitalInputs".sFrontDoorClosed.sSWStatus;
       "DB_OPC_RealTime".InfeedReadyOkStart := "DB_DigitalInputs".sInfeedReadyOK_Start.sSWStatus;
       "DB_OPC_RealTime".CoolingOK := "DB_DigitalInputs".sCoolingOK.sSWStatus;
       "DB_OPC_RealTime".PowerReady := "DB_DigitalInputs".sPowerReady.sSWStatus;
       "DB_OPC_RealTime".AlarmI2T := "DB_DigitalInputs".sAlarmI2T.sSWStatus;
       "DB_OPC_RealTime".HeadLaserBusy := "DB_DigitalInputs".sHeadLaserBusy.sSWStatus;
       "DB_OPC_RealTime".HeadLaserBreaker := "DB_DigitalInputs".sHeadLaserBreaker.sSWStatus;
       "DB_OPC_RealTime".FrontDoorLocked := "DB_DigitalInputs".sFrontDoorLocked.sSWStatus;
       "DB_OPC_RealTime".UPS_CommonAlarm := "DB_DigitalInputs".sUPS_CommonAlarm.sSWStatus;
       "DB_OPC_RealTime".UPS_BatteryLow := "DB_DigitalInputs".sUPS_BatteryLow.sSWStatus;
       "DB_OPC_RealTime".HeadChillerHighPressure := "DB_DigitalInputs".sHeadChillerHighPressure.sSWStatus;
       "DB_OPC_RealTime".HeadChillerWaterTemperature := "DB_DigitalInputs".sHeadChillerWaterTemperature.sSWStatus;
       "DB_OPC_RealTime".HeadChillerFlow := "DB_DigitalInputs".sHeadChillerFlow.sSWStatus;
       "DB_OPC_RealTime".HeadChillerCollectivFault := "DB_DigitalInputs".sHeadChillerCollectivFault.sSWStatus;
       "DB_OPC_RealTime".HeadChillerWaterLevel := "DB_DigitalInputs".sHeadChillerWaterLevel.sSWStatus;
       "DB_OPC_RealTime".UpsByPassActive := "DB_DigitalInputs".sUPS_ByPassActive.sSWStatus;
       "DB_OPC_RealTime".HeadChillerAmbiantTemperature := "DB_DigitalInputs".sHeadChillerAmbiantTemperature.sSWStatus;
       "DB_OPC_RealTime".LoadClampOpened := "DB_DigitalInputs".sLoadClampOpened.sSWStatus;
       "DB_OPC_RealTime".LoadClampNotClosedWithPart := "DB_DigitalInputs".sLoadClampNotClosedWithPart.sSWStatus;
       "DB_OPC_RealTime".UnloadClampOpened := "DB_DigitalInputs".sUnloadClampOpened.sSWStatus;
       "DB_OPC_RealTime".UpsFault := "DB_DigitalInputs".sUPS_Fault.sSWStatus;
       "DB_OPC_RealTime".InternalGateLocked := "DB_DigitalInputs".sInternalGateLocked.sSWStatus;
       "DB_OPC_RealTime".ExternalGateLocked := "DB_DigitalInputs".sExternalGateLocked.sSWStatus;
       "DB_OPC_RealTime".InverterActive := "DB_DigitalInputs".sInverterActive.sSWStatus;
       "DB_OPC_RealTime".UnloadClampNotClosedWithPart := "DB_DigitalInputs".sUnloadClampNotClosedWithPart.sSWStatus;
       "DB_OPC_RealTime".InternalGateOpened := "DB_DigitalInputs".sInternalGateOpened.sSWStatus;
       "DB_OPC_RealTime".ExternalGateOpened := "DB_DigitalInputs".sExternalGateOpened.sSWStatus;
       "DB_OPC_RealTime".PowerMeterBackCtrl := "DB_DigitalInputs".sPowerMeterBackCtrl.sSWStatus;
       "DB_OPC_RealTime".PowerMeterFrontCtrl := "DB_DigitalInputs".sPowerMeterFrontCtrl.sSWStatus;
       "DB_OPC_RealTime".HeadChillerCutOff := "DB_DigitalInputs".sHeadChillerCutOff.sSWStatus;
       "DB_OPC_RealTime".HeadChillerTemperature := "DB_DigitalInputs".sHeadChillerTemperature.sSWStatus;
       "DB_OPC_RealTime".ClampingOpenCtrl := "DB_DigitalInputs".sClampingOpenCtrl.sSWStatus;
       "DB_OPC_RealTime".B_AxisBrakeReleasedCtrl := "DB_DigitalInputs".sB_Axis_BrakeReleasedCtrl.sSWStatus;
       "DB_OPC_RealTime".B_AxisReferencePoint := "DB_DigitalInputs".sB_AxisReferencePoint.sSWStatus;
       "DB_OPC_RealTime".SourceChillerHighPressure := "DB_DigitalInputs".sSourceChillerHighPressure.sSWStatus;
       "DB_OPC_RealTime".SourceChillerWaterTemperature := "DB_DigitalInputs".sSourceChillerWaterTemperature.sSWStatus;
       "DB_OPC_RealTime".SourceChillerFlow := "DB_DigitalInputs".sSourceChillerFlow.sSWStatus;
       "DB_OPC_RealTime".SourceChillerCollectivFault := "DB_DigitalInputs".sSourceChillerCollectivFault.sSWStatus;
       "DB_OPC_RealTime".SourceChillerWaterLevel := "DB_DigitalInputs".sSourceChillerWaterLevel.sSWStatus;
       "DB_OPC_RealTime".SourceChillerAmbiantTemperature := "DB_DigitalInputs".sSourceChillerAmbiantTemperature.sSWStatus;
       "DB_OPC_RealTime".SourceChillerCutOff := "DB_DigitalInputs".sSourceChillerCutOff.sSWStatus;
       "DB_OPC_RealTime".SourceChillerTemperature := "DB_DigitalInputs".sSourceChillerTemperature.sSWStatus;
   END_REGION

   REGION Digital Outputs
       "DB_OPC_RealTime".OperatingCounter := "DB_DigitalOutputs".sOperatingCounter.sSWStatus;
       "DB_OPC_RealTime".GeneralAirValve := "DB_DigitalOutputs".sGeneralAirValve.sSWStatus;
       "DB_OPC_RealTime".SmartLineDisable := "DB_DigitalOutputs".sSmartLineDisable.sSWStatus;
       "DB_OPC_RealTime".MachineLight := "DB_DigitalOutputs".sMachineLight.sSWStatus;
       "DB_OPC_RealTime".MachineLightBack := "DB_DigitalOutputs".sMachineLightBack.sSWStatus;
       "DB_OPC_RealTime".LightTowerOrange := "DB_DigitalOutputs".sLightTowerOrange.sSWStatus;
       "DB_OPC_RealTime".LightTowerRed := "DB_DigitalOutputs".sLightTowerRed.sSWStatus;
       "DB_OPC_RealTime".LightTowerBlue := "DB_DigitalOutputs".sLightTowerBlue.sSWStatus;
       "DB_OPC_RealTime".LightTowerGreen := "DB_DigitalOutputs".sLightTowerGreen.sSWStatus;
       "DB_OPC_RealTime".LightTowerWhite := "DB_DigitalOutputs".sLightTowerWhite.sSWStatus;
       "DB_OPC_RealTime".Backlight := "DB_DigitalOutputs".sBacklight.sSWStatus;
       "DB_OPC_RealTime".InfeedON := "DB_DigitalOutputs".sInfeedON.sSWStatus;
       "DB_OPC_RealTime".AxisActivation := "DB_DigitalOutputs".sAxisActivation.sSWStatus;
       "DB_OPC_RealTime".BuzzerActivation := "DB_DigitalOutputs".sBuzzerActivation.sSWStatus;
       "DB_OPC_RealTime".ElbaronPowerON := "DB_DigitalOutputs".sElbaronPowerON.sSWStatus;
       "DB_OPC_RealTime".ObservationCameraLight := "DB_DigitalOutputs".sObservationCameraLight.sSWStatus;
       "DB_OPC_RealTime".LaserExternalDoorOpening := "DB_DigitalOutputs".sLaserExternalDoorOpening.sSWStatus;
       "DB_OPC_RealTime".CoolingStart := "DB_DigitalOutputs".sCoolingStart.sSWStatus;
       "DB_OPC_RealTime".X_AxisBrakeActivation := "DB_DigitalOutputs".sX_AxisBrakeActivation.sSWStatus;
       "DB_OPC_RealTime".Y_AxisBrakeActivation := "DB_DigitalOutputs".sY_AxisBrakeActivation.sSWStatus;
       "DB_OPC_RealTime".AxisB_TeachInClampingPart := "DB_DigitalOutputs".sAxisB_TeachInClampingPart.sSWStatus;
       "DB_OPC_RealTime".EPO_UPS := "DB_DigitalOutputs".sEPO_UPS.sSWStatus;
       "DB_OPC_RealTime".HeadLaserStart := "DB_DigitalOutputs".sHeadLaserStart.sSWStatus;
       "DB_OPC_RealTime".HeadLaserStop := "DB_DigitalOutputs".sHeadLaserStop.sSWStatus;
       "DB_OPC_RealTime".Axis2_PowerContactor := "DB_DigitalOutputs".sAxis2_PowerContactor.sSWStatus;
       "DB_OPC_RealTime".GasAssistOn := "DB_DigitalOutputs".sGasAssistOn.sSWStatus;
       "DB_OPC_RealTime".SmartLineReset := "DB_DigitalOutputs".sSmartLineReset.sSWStatus;
       "DB_OPC_RealTime".XY_AxisPowerContactor := "DB_DigitalOutputs".sXY_AxisPowerContactor.sSWStatus;
       "DB_OPC_RealTime".LaserAirPressureProcess := "DB_DigitalOutputs".sLaserAirPressureProcess.sSWStatus;
       "DB_OPC_RealTime".Bus60V_PowerContactor := "DB_DigitalOutputs".sBus60V_PowerContactor.sSWStatus;
       "DB_OPC_RealTime".LoadClampClosing := "DB_DigitalOutputs".sLoadClampClosing.sSWStatus;
       "DB_OPC_RealTime".LoadClampOpening := "DB_DigitalOutputs".sLoadClampOpening.sSWStatus;
       "DB_OPC_RealTime".UnloadClampClosing := "DB_DigitalOutputs".sUnloadClampClosing.sSWStatus;
       "DB_OPC_RealTime".UnloadClampOpening := "DB_DigitalOutputs".sUnloadClampOpening.sSWStatus;
       "DB_OPC_RealTime".ClampingOpening := "DB_DigitalOutputs".sClampingOpening.sSWStatus;
       "DB_OPC_RealTime".ClampingClosing := "DB_DigitalOutputs".sClampingClosing.sSWStatus;
       "DB_OPC_RealTime".B_AxisBrakeRelease := "DB_DigitalOutputs".sB_AxisBrakeRelease.sSWStatus;
       "DB_OPC_RealTime".Suction := "DB_DigitalOutputs".sSuction.sSWStatus;
       "DB_OPC_RealTime".ExternalGateClosing := "DB_DigitalOutputs".sExternalGateClosing.sSWStatus;
       "DB_OPC_RealTime".ExternalGateOpening := "DB_DigitalOutputs".sExternalGateOpening.sSWStatus;
       "DB_OPC_RealTime".InternalGateClosing := "DB_DigitalOutputs".sInternalGateClosing.sSWStatus;
       "DB_OPC_RealTime".InternalGateOpening := "DB_DigitalOutputs".sInternalGateOpening.sSWStatus;
       "DB_OPC_RealTime".PowerMeterRetract := "DB_DigitalOutputs".sPowerMeterRetract.sSWStatus;
       "DB_OPC_RealTime".PowerMeterAdvance := "DB_DigitalOutputs".sPowerMeterAdvance.sSWStatus;
       "DB_OPC_RealTime".Blowing := "DB_DigitalOutputs".sBlowing.sSWStatus;
   END_REGION

   REGION Analog Inputs
       "DB_OPC_RealTime".LaserPowerMeter := "DB_AnalogInputs".sLaserPowerMeter.sSWRealValue;
       "DB_OPC_RealTime".AxisB_ClampingPart := "DB_AnalogInputs".sAxisB_ClampingPart.sSWRealValue;
       "DB_OPC_RealTime".LaserAirPressureProcess_1 := "DB_AnalogInputs".sLaserAirPressureProcess.sSWRealValue;
       "DB_OPC_RealTime".InletAirPressure := "DB_AnalogInputs".sInletAirPressure.sSWRealValue;
       "DB_OPC_RealTime".AmbiantTemperature := "DB_AnalogInputs".sAmbiantTemperature.sSWRealValue;
       "DB_OPC_RealTime".MachineTemperature := "DB_AnalogInputs".sMachineTemperature.sSWRealValue;
       "DB_OPC_RealTime".Cold_WaterTemperatureInput := "DB_AnalogInputs".sCold_WaterTemperatureInput.sSWRealValue;
       "DB_OPC_RealTime".Cold_WaterTemperatureOutput := "DB_AnalogInputs".sCold_WaterTemperatureOutput.sSWRealValue;
       "DB_OPC_RealTime".X_AxisTemperaturePT1000 := "DB_AnalogInputs".sX_AxisTemperaturePT1000.sSWRealValue;
       "DB_OPC_RealTime".Y_AxisTemperaturePT1000 := "DB_AnalogInputs".sY_AxisTemperaturePT1000.sSWRealValue;
       "DB_OPC_RealTime".X_AxisTemperaturePTC := "DB_AnalogInputs".sX_AxisTemperaturePTC.sSWRealValue;
       "DB_OPC_RealTime".Y_AxisTemperaturePTC := "DB_AnalogInputs".sY_AxisTemperaturePTC.sSWRealValue;
       "DB_OPC_RealTime".NozzleOverpressure := "DB_AnalogInputs".sNozzleOverpressure.sSWRealValue;
       "DB_OPC_RealTime".OpticalPathOverpressure := "DB_AnalogInputs".sOpticalPathOverpressure.sSWRealValue;
       "DB_OPC_RealTime".LaserHeadOverpressure := "DB_AnalogInputs".sLaserHeadOverpressure.sSWRealValue;
       "DB_OPC_RealTime".ZLAxisOverpressure := "DB_AnalogInputs".sZLAxisOverpressure.sSWRealValue;
       "DB_OPC_RealTime".XYAxisOverpressure := "DB_AnalogInputs".sXYAxisOverpressure.sSWRealValue;
       "DB_OPC_RealTime".LeftAspiration := "DB_AnalogInputs".sLeftAspiration.sSWRealValue;
       "DB_OPC_RealTime".RightAspiration := "DB_AnalogInputs".sRightAspiration.sSWRealValue;
       "DB_OPC_RealTime".ClimTemperature := "DB_AnalogInputs".sClimTemperature.sSWRealValue;
       "DB_OPC_RealTime".SensorControllerStation1 := "DB_AnalogInputs".sSensorControllerStation1.sSWRealValue;
       "DB_OPC_RealTime".CabinetTemperature := "DB_AnalogInputs".sCabinetTemperature.sSWRealValue;
   END_REGION

   REGION Analog Outputs
       "DB_OPC_RealTime".NozzleOverpressureSetPoint := "DB_AnalogOutputs".sNozzleOverpressureSetPoint.sSWRealValue;
       "DB_OPC_RealTime".VentilatorSetPoint := "DB_AnalogOutputs".sVentilatorSetPoint.sSWRealValue;
       "DB_OPC_RealTime".PropValveClimSetPoint := "DB_AnalogOutputs".sPropValveClimSetPoint.sSWRealValue;
   END_REGION
END_FUNCTION_BLOCK

FUNCTION_BLOCK "FB_Components"   // FB83, SCL
{ S7_Optimized_Access := 'TRUE' }
// stored: MemoryReserve 100, SetENOAutomatically false
   VAR
      sRT_Update : R_TRIG;
      sShuttle1DrilledPart : "FB_OPC_PartStatus";
      sShuttle1UndrilledPart { S7_SetPoint := 'True'} : "FB_OPC_PartStatus";
      sShuttle2DrilledPart { S7_SetPoint := 'True'} : "FB_OPC_PartStatus";
      sShuttle2UndrilledPart { S7_SetPoint := 'True'} : "FB_OPC_PartStatus";
      sShuttle1DrilledBw : "FB_OPC_PartStatus";
      sShuttle1UndrilledBw { S7_SetPoint := 'True'} : "FB_OPC_PartStatus";
      sShuttle2DrilledBw { S7_SetPoint := 'True'} : "FB_OPC_PartStatus";
      sShuttle2UndrilledBw { S7_SetPoint := 'True'} : "FB_OPC_PartStatus";
      sGripperDrilledPart : "FB_OPC_PartStatus";
      sGripperUndrilledPart { S7_SetPoint := 'True'} : "FB_OPC_PartStatus";
      sGripperDrilledBw : "FB_OPC_PartStatus";
      sGripperUndrilledBw { S7_SetPoint := 'True'} : "FB_OPC_PartStatus";
      sFixtureDrilledPart : "FB_OPC_PartStatus";
      sFixtureUndrilledPart { S7_SetPoint := 'True'} : "FB_OPC_PartStatus";
      sFixtureDrilledBw : "FB_OPC_PartStatus";
      sFixtureUndrilledBw { S7_SetPoint := 'True'} : "FB_OPC_PartStatus";
   END_VAR
BEGIN
   REGION Description header 
       //==================================================================================
       // POSALUX Swiss SA / (C) Copyright 2026
       //----------------------------------------------------------------------------------
       // Title: FB_Components
       // Comment/Function: 
       //
       // Author: Fabien WALDT
       // Engineering: TIA Portal v20
       //----------------------------------------------------------------------------------
       // Change log table:
       // Version  | Date     | Expert in charge | Changes applied
       // ---------|----------|------------------|------------------------------------
       // 00.00.01 | 20260310 | WFA              | First released version
       // ==================================================================================
   END_REGION

   REGION Shuttle 1
       // Drilled Part
       #sShuttle1DrilledPart(iGood := "DB_PartManagement".sPosition.sShuttle1.Drilled.States.Part.Good,
                             iUnknown := "DB_PartManagement".sPosition.sShuttle1.Drilled.States.Part.Unknown,
                             iBad := "DB_PartManagement".sPosition.sShuttle1.Drilled.States.Part.Bad,
                             iAbsent := "DB_PartManagement".sPosition.sShuttle1.Drilled.States.Part.Absent,
                             iPresentUnexpected := "DB_PartManagement".sPosition.sShuttle1.Drilled.States.Part.PresentUnexpected,
                             iAbsentUnexpected := "DB_PartManagement".sPosition.sShuttle1.Drilled.States.Part.AbsentUnexpected,
                             oStatus => "DB_OPC_Components".Parts.ShuttleDrilled);

       // Undrilled Part
       #sShuttle1UndrilledPart(iGood := "DB_PartManagement".sPosition.sShuttle1.Undrilled.States.Part.Good,
                               iUnknown := "DB_PartManagement".sPosition.sShuttle1.Undrilled.States.Part.Unknown,
                               iBad := "DB_PartManagement".sPosition.sShuttle1.Undrilled.States.Part.Bad,
                               iAbsent := "DB_PartManagement".sPosition.sShuttle1.Undrilled.States.Part.Absent,
                               iPresentUnexpected := "DB_PartManagement".sPosition.sShuttle1.Undrilled.States.Part.PresentUnexpected,
                               iAbsentUnexpected := "DB_PartManagement".sPosition.sShuttle1.Undrilled.States.Part.AbsentUnexpected,
                               oStatus => "DB_OPC_Components".Parts.ShuttleUndrilled);
         // Drilled Bw
       #sShuttle1DrilledBw(iGood := "DB_PartManagement".sPosition.sShuttle1.Drilled.States.BW.Good,
                           iUnknown := "DB_PartManagement".sPosition.sShuttle1.Drilled.States.BW.Unknown,
                           iBad := "DB_PartManagement".sPosition.sShuttle1.Drilled.States.BW.Bad,
                           iAbsent := "DB_PartManagement".sPosition.sShuttle1.Drilled.States.BW.Absent,
                           iPresentUnexpected := "DB_PartManagement".sPosition.sShuttle1.Drilled.States.BW.PresentUnexpected,
                           iAbsentUnexpected := "DB_PartManagement".sPosition.sShuttle1.Drilled.States.BW.AbsentUnexpected,
                           oStatus => "DB_OPC_Components".Backwalls.ShuttleDrilled);

         // Undrilled Bw
       #sShuttle1UndrilledBw(iGood := "DB_PartManagement".sPosition.sShuttle1.Undrilled.States.BW.Good,
                             iUnknown := "DB_PartManagement".sPosition.sShuttle1.Undrilled.States.BW.Unknown,
                             iBad := "DB_PartManagement".sPosition.sShuttle1.Undrilled.States.BW.Bad,
                             iAbsent := "DB_PartManagement".sPosition.sShuttle1.Undrilled.States.BW.Absent,
                             iPresentUnexpected := "DB_PartManagement".sPosition.sShuttle1.Undrilled.States.BW.PresentUnexpected,
                             iAbsentUnexpected := "DB_PartManagement".sPosition.sShuttle1.Undrilled.States.BW.AbsentUnexpected,
                             oStatus => "DB_OPC_Components".Backwalls.ShuttleUndrilled);
   END_REGION

   REGION Shuttle 2
       // Drilled Part
       #sShuttle2DrilledPart(iGood := "DB_PartManagement".sPosition.sShuttle2.Drilled.States.Part.Good,
                             iUnknown := "DB_PartManagement".sPosition.sShuttle2.Drilled.States.Part.Unknown,
                             iBad := "DB_PartManagement".sPosition.sShuttle2.Drilled.States.Part.Bad,
                             iAbsent := "DB_PartManagement".sPosition.sShuttle2.Drilled.States.Part.Absent,
                             iPresentUnexpected := "DB_PartManagement".sPosition.sShuttle2.Drilled.States.Part.PresentUnexpected,
                             iAbsentUnexpected := "DB_PartManagement".sPosition.sShuttle2.Drilled.States.Part.AbsentUnexpected,
                             oStatus => "DB_OPC_Components".Parts.Shuttle2Drilled);

       // Undrilled Part
       #sShuttle2UndrilledPart(iGood := "DB_PartManagement".sPosition.sShuttle2.Undrilled.States.Part.Good,
                               iUnknown := "DB_PartManagement".sPosition.sShuttle2.Undrilled.States.Part.Unknown,
                               iBad := "DB_PartManagement".sPosition.sShuttle2.Undrilled.States.Part.Bad,
                               iAbsent := "DB_PartManagement".sPosition.sShuttle2.Undrilled.States.Part.Absent,
                               iPresentUnexpected := "DB_PartManagement".sPosition.sShuttle2.Undrilled.States.Part.PresentUnexpected,
                               iAbsentUnexpected := "DB_PartManagement".sPosition.sShuttle2.Undrilled.States.Part.AbsentUnexpected,
                               oStatus => "DB_OPC_Components".Parts.Shuttle2Undrilled);
       // Drilled Bw
       #sShuttle2DrilledBw(iGood := "DB_PartManagement".sPosition.sShuttle2.Drilled.States.BW.Good,
                           iUnknown := "DB_PartManagement".sPosition.sShuttle2.Drilled.States.BW.Unknown,
                           iBad := "DB_PartManagement".sPosition.sShuttle2.Drilled.States.BW.Bad,
                           iAbsent := "DB_PartManagement".sPosition.sShuttle2.Drilled.States.BW.Absent,
                           iPresentUnexpected := "DB_PartManagement".sPosition.sShuttle2.Drilled.States.BW.PresentUnexpected,
                           iAbsentUnexpected := "DB_PartManagement".sPosition.sShuttle2.Drilled.States.BW.AbsentUnexpected,
                           oStatus => "DB_OPC_Components".Backwalls.Shuttle2Drilled);

       // Undrilled Bw
       #sShuttle2UndrilledBw(iGood := "DB_PartManagement".sPosition.sShuttle2.Undrilled.States.BW.Good,
                             iUnknown := "DB_PartManagement".sPosition.sShuttle2.Undrilled.States.BW.Unknown,
                             iBad := "DB_PartManagement".sPosition.sShuttle2.Undrilled.States.BW.Bad,
                             iAbsent := "DB_PartManagement".sPosition.sShuttle2.Undrilled.States.BW.Absent,
                             iPresentUnexpected := "DB_PartManagement".sPosition.sShuttle2.Undrilled.States.BW.PresentUnexpected,
                             iAbsentUnexpected := "DB_PartManagement".sPosition.sShuttle2.Undrilled.States.BW.AbsentUnexpected,
                             oStatus => "DB_OPC_Components".Backwalls.Shuttle2Undrilled);
   END_REGION

   REGION Gripper
       // Drilled Part
       #sGripperDrilledPart(iGood := "DB_PartManagement".sPosition.sGripper.Drilled.States.Part.Good,
                            iUnknown := "DB_PartManagement".sPosition.sGripper.Drilled.States.Part.Unknown,
                            iBad := "DB_PartManagement".sPosition.sGripper.Drilled.States.Part.Bad,
                            iAbsent := "DB_PartManagement".sPosition.sGripper.Drilled.States.Part.Absent,
                            iPresentUnexpected :=  "DB_PartManagement".sPosition.sGripper.Drilled.States.Part.PresentUnexpected,
                            iAbsentUnexpected := "DB_PartManagement".sPosition.sGripper.Drilled.States.Part.AbsentUnexpected,
                            oStatus => "DB_OPC_Components".Parts.LoaderDrilled);

       // Undrilled Part
       #sGripperUndrilledPart(iGood := "DB_PartManagement".sPosition.sGripper.Undrilled.States.Part.Good,
                              iUnknown := "DB_PartManagement".sPosition.sGripper.Undrilled.States.Part.Unknown,
                              iBad := "DB_PartManagement".sPosition.sGripper.Undrilled.States.Part.Bad,
                              iAbsent := "DB_PartManagement".sPosition.sGripper.Undrilled.States.Part.Absent,
                              iPresentUnexpected :=  "DB_PartManagement".sPosition.sGripper.Undrilled.States.Part.PresentUnexpected,
                              iAbsentUnexpected := "DB_PartManagement".sPosition.sGripper.Undrilled.States.Part.AbsentUnexpected,
                              oStatus => "DB_OPC_Components".Parts.LoaderUndrilled);
       // Drilled Bw
       #sGripperDrilledBw(iGood := "DB_PartManagement".sPosition.sGripper.Drilled.States.BW.Good,
                          iUnknown := "DB_PartManagement".sPosition.sGripper.Drilled.States.BW.Unknown,
                          iBad := "DB_PartManagement".sPosition.sGripper.Drilled.States.BW.Bad,
                          iAbsent := "DB_PartManagement".sPosition.sGripper.Drilled.States.BW.Absent,
                          iPresentUnexpected :=  "DB_PartManagement".sPosition.sGripper.Drilled.States.BW.PresentUnexpected,
                          iAbsentUnexpected := "DB_PartManagement".sPosition.sGripper.Drilled.States.BW.AbsentUnexpected,
                          oStatus => "DB_OPC_Components".Backwalls.LoaderDrilled);

       // Undrilled Bw
       #sGripperUndrilledBw(iGood := "DB_PartManagement".sPosition.sGripper.Undrilled.States.BW.Good,
                            iUnknown := "DB_PartManagement".sPosition.sGripper.Undrilled.States.BW.Unknown,
                            iBad := "DB_PartManagement".sPosition.sGripper.Undrilled.States.BW.Bad,
                            iAbsent := "DB_PartManagement".sPosition.sGripper.Undrilled.States.BW.Absent,
                            iPresentUnexpected :=  "DB_PartManagement".sPosition.sGripper.Undrilled.States.BW.PresentUnexpected,
                            iAbsentUnexpected := "DB_PartManagement".sPosition.sGripper.Undrilled.States.BW.AbsentUnexpected,
                            oStatus => "DB_OPC_Components".Backwalls.LoaderUndrilled);
                         END_REGION

   REGION Fixture
     // Drilled - Undrilled Part
       #sFixtureDrilledPart(iGood := "DB_PartManagement".sPosition.sFixture.Drilled.States.Part.Good OR "DB_PartManagement".sPosition.sFixture.Undrilled.States.Part.Good,
                            iUnknown := "DB_PartManagement".sPosition.sFixture.Drilled.States.Part.Unknown,
                            iBad := "DB_PartManagement".sPosition.sFixture.Drilled.States.Part.Bad,
                            iAbsent := "DB_PartManagement".sPosition.sFixture.Drilled.States.Part.Absent,
                            iPresentUnexpected := "DB_PartManagement".sPosition.sFixture.Drilled.States.Part.PresentUnexpected,
                            iAbsentUnexpected := "DB_PartManagement".sPosition.sFixture.Drilled.States.Part.AbsentUnexpected,
                            oStatus => "DB_OPC_Components".Parts.WorkClamp);

     // Drilled Bw
       #sFixtureDrilledBw(iGood := "DB_PartManagement".sPosition.sFixture.Drilled.States.BW.Good OR "DB_PartManagement".sPosition.sFixture.Undrilled.States.BW.Good,
                          iUnknown := "DB_PartManagement".sPosition.sFixture.Drilled.States.BW.Unknown,
                          iBad := "DB_PartManagement".sPosition.sFixture.Drilled.States.BW.Bad,
                          iAbsent := "DB_PartManagement".sPosition.sFixture.Drilled.States.BW.Absent,
                          iPresentUnexpected := "DB_PartManagement".sPosition.sFixture.Drilled.States.BW.PresentUnexpected,
                          iAbsentUnexpected := "DB_PartManagement".sPosition.sFixture.Drilled.States.BW.AbsentUnexpected,
                          oStatus => "DB_OPC_Components".Backwalls.WorkClamp);
   END_REGION

   REGION Update
       #sRT_Update(CLK := "Clock_1Hz");
       IF #sRT_Update.Q THEN
           "DB_OPC_Components".Update := "DB_OPC_Components".Update + 1;
       END_IF;

       IF "DB_OPC_Components".Update >= 255 THEN
           "DB_OPC_Components".Update := 0;
       END_IF;
   END_REGION
END_FUNCTION_BLOCK

FUNCTION_BLOCK "FB_OPC_PartStatus"   // FB47, SCL
{ S7_Optimized_Access := 'TRUE' }
// stored: MemoryReserve 100, SetENOAutomatically false
   VAR_INPUT
      iGood { ExternalAccessible := 'False'; ExternalVisible := 'False'; ExternalWritable := 'False'} : Bool;
      iUnknown { ExternalAccessible := 'False'; ExternalVisible := 'False'; ExternalWritable := 'False'} : Bool;
      iBad { ExternalAccessible := 'False'; ExternalVisible := 'False'; ExternalWritable := 'False'} : Bool;
      iAbsent { ExternalAccessible := 'False'; ExternalVisible := 'False'; ExternalWritable := 'False'} : Bool;
      iPresentUnexpected { ExternalAccessible := 'False'; ExternalVisible := 'False'; ExternalWritable := 'False'} : Bool;
      iAbsentUnexpected { ExternalAccessible := 'False'; ExternalVisible := 'False'; ExternalWritable := 'False'} : Bool;
   END_VAR
   VAR_OUTPUT
      oStatus { ExternalAccessible := 'False'; ExternalVisible := 'False'; ExternalWritable := 'False'} : Byte;
   END_VAR
   VAR CONSTANT
      GOOD : Byte := 3;
      UNKNOW : Byte := 1;
      BAD : Byte := 2;
      ABSENT : Byte := 0;
      PRESENT_UNEXPECTED : Byte := 4;
      ABSENT_UNEXPECTED : Byte := 5;
      UNKNOW_STATUS : Byte := 99;
   END_VAR
BEGIN
   REGION Description header 
       //==================================================================================
       // POSALUX Swiss SA / (C) Copyright 2024
       //----------------------------------------------------------------------------------
       // Title: 
       // Comment/Function: 
       //
       // Author: Fabien WALDT
       // Engineering: TIA Portal v20
       //----------------------------------------------------------------------------------
       // Change log table:
       // Version  | Date     | Expert in charge | Changes applied
       // ---------|----------|------------------|------------------------------------
       // 00.00.01 | 20251024 | WFA              | First released version
       // ==================================================================================
   END_REGION

   REGION Status
       IF #iGood THEN
           #oStatus := #GOOD;
       ELSIF #iUnknown THEN
           #oStatus := #UNKNOW;
       ELSIF #iBad THEN
           #oStatus := #BAD;
       ELSIF #iAbsent THEN
           #oStatus := #ABSENT;
       ELSIF #iPresentUnexpected THEN
           #oStatus := #PRESENT_UNEXPECTED;
       ELSIF #iAbsentUnexpected THEN
           #oStatus := #ABSENT_UNEXPECTED;
       ELSE
           #oStatus := #UNKNOW_STATUS;
       END_IF;
   END_REGION
END_FUNCTION_BLOCK

FUNCTION_BLOCK "FB_Scanner"   // FB89, SCL
{ S7_Optimized_Access := 'TRUE' }
// stored: MemoryReserve 100, SetENOAutomatically false
   VAR
      sScannerComm : "FB_ScannerComm";
      sReadR_Param { S7_SetPoint := 'True'} : "LBP_ReadVar";
      sWriteR_Param { S7_SetPoint := 'True'} : "LBP_WriteVar";
      sError { ExternalAccessible := 'False'; ExternalVisible := 'False'; ExternalWritable := 'False'} : Bool;
      sNDR { ExternalAccessible := 'False'; ExternalVisible := 'False'; ExternalWritable := 'False'} : Bool;
      sState { ExternalAccessible := 'False'; ExternalVisible := 'False'; ExternalWritable := 'False'} : Word;
      sR94 : LReal;
      sR95 : LReal;
      sR96 : LReal;
      sR97 : LReal;
      sJobNamePart : DInt;
      sJobNamePowerMeter : DInt;
      sMeasureZ : LReal;
      sVarName { S7_SetPoint := 'True'} : String;
      sReadGUD_JobNamePart { S7_SetPoint := 'True'} : "LBP_ReadGUD";
      sReadGUD_JobNamePowerMeter { S7_SetPoint := 'True'} : "LBP_ReadGUD";
      sReadGUD_MeasureZ { S7_SetPoint := 'True'} : "LBP_ReadGUD";
      sWriteR_ParamReq { S7_SetPoint := 'True'} : Bool;
      sTimePulseWriteParam : TON_TIME;
   END_VAR
BEGIN
   REGION Description header 
       //==================================================================================
       // POSALUX Swiss SA / (C) Copyright 2026
       //----------------------------------------------------------------------------------
       // Title: FB_Scanner
       // Comment/Function: 
       //
       // Author: Fabien WALDT
       // Engineering: TIA Portal v20
       //----------------------------------------------------------------------------------
       // Change log table:
       // Version  | Date     | Expert in charge | Changes applied
       // ---------|----------|------------------|------------------------------------
       // 00.00.01 | 20260330 | WFA              | First released version
       // ==================================================================================
   END_REGION

   REGION NC Exchanges
       // Job Request
       #sReadR_Param(Req := "Clock_10Hz" AND NOT  #sWriteR_Param.Req,
                                NumVar := 4,
                                Addr1 := "DB_NcVarSelect_R_Param"."$R[96]".token,
                                Addr2 := "DB_NcVarSelect_R_Param"."$R[97]".token,
                                Addr3 := "DB_NcVarSelect_R_Param"."$R[95]".token,
                                Addr4 := "DB_NcVarSelect_R_Param"."$R[94]".token,
                                Addr5 := NULL,
                                Addr6 := NULL,
                                Addr7 := NULL,
                                Addr8 := NULL,
                                Error => #sError,
                                NDR => #sNDR,
                                State => #sState,
                                RD1 := #sR96,
                                RD2 := #sR97,
                                RD3 := #sR95,
                                RD4 := #sR94,
                                RD5 := NULL,
                                RD6 := NULL,
                                RD7 := NULL,
                                RD8 := NULL);

                  #sWriteR_Param(Req := #sWriteR_ParamReq AND NOT #sReadR_Param.Req,
                                 NumVar := 3,
                                 Addr1 := "DB_NcVarSelect_R_Param"."$R[96]".token,
                                 Addr2 := "DB_NcVarSelect_R_Param"."$R[97]".token,
                                 Addr3 := "DB_NcVarSelect_R_Param"."$R[95]".token,
                                 Addr4 := NULL,
                                 Addr5 := NULL,
                                 Addr6 := NULL,
                                 Addr7 := NULL,
                                 Addr8 := NULL,
                                 Error => #sError,
                                 Done => #sNDR,
                                 State => #sState,
                                 SD1 := #sR96,
                                 SD2 := #sR97,
                                 SD3 := #sR95,
                                 SD4 := NULL,
                                 SD5 := NULL,
                                 SD6 := NULL,
                                 SD7 := NULL,
                                 SD8 := NULL);

       // RequestJob
       // Job request if R96 <> 0 and R97 = 0
       #sScannerComm.ioRequestJob_NC := #sR96 <> 0 AND #sR97 = 0;

       // Station Number
           // Si powermeter not IN Station = 0 
           IF NOT "DB_DigitalInputs".sPowerMeterBackCtrl.sSWStatus THEN
               #sScannerComm.iStationNumber := 0;
           ELSE
               #sScannerComm.iStationNumber := 1;
           END_IF;

       // Hole Number
           #sScannerComm.iHoleNumber := LREAL_TO_DINT(#sR95);

       // Job list Name
           // Variable écrite dans FB_Recipe
       // Job Name
            // Job Name Part
           #sVarName := 'H_J';

           #sReadGUD_JobNamePart(Req := "Clock_1Hz",
                              Addr := #sVarName,
                              Area := 2,
                              Unit := 1,
                              Index1 := 0,
                              Index2 := 1,
                              CnvtToken := FALSE,
                              VarToken := NULL,
                              Error => #sReadGUD_JobNamePart.Error,
                              Done => #sReadGUD_JobNamePart.Done,
                              State => #sReadGUD_JobNamePart.State,
                              RD := #sJobNamePart);

        // Job Name Part
        #sVarName := 'L_P_J';

        #sReadGUD_JobNamePowerMeter(Req := "Clock_1Hz",
                                    Addr := #sVarName,
                                    Area := 0,
                                    Unit := 1,
                                    Index1 := 1,
                                    Index2 := 0,
                                    CnvtToken := FALSE,
                                    VarToken := NULL,
                                    Error => #sReadGUD_JobNamePowerMeter.Error,
                                    Done => #sReadGUD_JobNamePowerMeter.Done,
                                    State => #sReadGUD_JobNamePowerMeter.State,
                                    RD := #sJobNamePowerMeter);

   IF #sScannerComm.iStationNumber = 0 THEN
       #sScannerComm.iJobName := #sJobNamePowerMeter;
   ELSE
       #sScannerComm.iJobName := #sJobNamePart;
   END_IF;

       // Measure Z
   #sMeasureZ := #sR94;
   END_REGION

